Staubli VAL3: Shell.dtx

bool b1 = true
bool b2 = true
bool bExit
bool bInit
bool bListRefresh = true
bool bPause
bool bRobAtStP
bool bUserRefresh = true
dio distart = {link=usrIn0}
dio distop = {link=usrIn1}
dio ditab = {link=BasicIO-1\%I1}
dio dixi = {link=BasicIO-1\%I0}
dio dochui = {link=BasicIO-1\%Q0}
dio doxi = {link=BasicIO-1\%Q1}
frame f1 = {x=118.3, y=-256.27, z=-98.22, rx=-0.18, ry=0.05, rz=179.93, fatherId=world[0]}
frame fFrmTemp = {x=480, y=75, z=-95.95, rx=5, ry=0, rz=-93, fatherId=world[0]}
frame frmaster = {x=480, y=75, z=-95.95, rx=5, rz=-93, fatherId=world[0]}
jointRx jXieLiao = {j1=-98.995401, j2=73.939591, j3=22.369301, j4=-0.0214, j5=83.505129, j6=-98.792613}
jointRx jbegin = {j1=-36.809158, j2=6.473103, j3=115.475326, j4=0.67904, j5=57.498227, j6=-129.910351}
jointRx jchack = {j1=-93.592762, j2=7.01746, j3=116.913403, j4=-0.052986, j5=55.884155, j6=86.700695}
jointRx jend = {j1=-46.642796, j2=10.279087, j3=109.084102, j4=6.799386, j5=57.689141, j6=-43.494821}
jointRx jready = {j1=-93.60071, j2=14.149819, j3=120.13944, j4=-0.061569, j5=45.526614, j6=86.705521}
jointRx jstart = {j1=-93.593066, j2=7.017202, j3=116.913452, j4=-0.053086, j5=55.884413, j6=86.699801}
mdesc m1
mdesc mSuDu[3]
  [0] = {leave=0.5, reach=0.5}
  [1] = {accel=25, vel=50, decel=25, leave=0.5, reach=0.5}
  [2] = {leave=0.5, reach=0.5}
num n0 = 1
num n1 = 2
num n2
num nBeltLifeTime = 1000
num nPY
num nPYB
num nPYC
num nPYtest
num nPage
num nSelected
num nSize = 314
num nc
num ndemo = 314
num ni
pointRx p1 = {x=0.29, y=-0.21, z=62.49, rx=-180, rz=179.71, fatherId=f1[0]}
pointRx p2 = {x=0.29, y=-0.21, z=-0.5, rx=-180, rz=179.71, fatherId=f1[0]}
pointRx p3 = {x=-135.757719, y=-14.921956, z=109.991113, rx=0.040194, ry=-179.896326, rz=-0.477597, fatherId=f1[0]}
pointRx p4 = {x=-342.629435, y=-93.502982, z=80.205763, rx=0.07546, ry=-170.514293, rz=20.52476, fatherId=f1[0]}
pointRx p5 = {x=-343.525561, y=-394.240354, z=80.654544, rx=173.283811, ry=-0.218212, rz=-67.079827, fatherId=f1[0]}
pointRx pTemp = {x=-72.136382, y=-5.208147, z=99.387825, rx=179.99914, ry=-2.97245, rz=-27.003129, shoulder=lefty, elbow=epositive, wrist=wpositive, fatherId=fFrmTemp[0]}
pointRx pXieLiao[2]
  [0] = {x=530.900904, y=-168.692362, z=119.392812, rx=179.999348, ry=-0.000559, rz=86.125781, fatherId=f1[0]}
  [1] = {x=530.900895, y=-168.692364, z=88.853022, rx=179.999359, ry=-0.000487, rz=86.125781, fatherId=f1[0]}
pointRx pdemo[900]
  [0] = {x=-72.139316, y=-5.205403, z=114.395923, rx=-179.99945, ry=-2.972824, rz=-27.002856, shoulder=lefty, elbow=epositive, wrist=wpositive, fatherId=frmaster[0]}
  [1] = {x=-72.141191, y=-5.207684, z=109.390059, rx=179.999959, ry=-2.973162, rz=-27.002729, shoulder=lefty, elbow=epositive, wrist=wpositive, fatherId=frmaster[0]}
  [2] = {x=-72.136382, y=-5.208147, z=99.387825, rx=179.99914, ry=-2.97245, rz=-27.003129, shoulder=lefty, elbow=epositive, wrist=wpositive, fatherId=frmaster[0]}
  [3] = {x=-68.975889, y=-15.06218, z=100.784201, rx=179.999892, ry=-4.176426, rz=-34.805987, shoulder=lefty, elbow=epositive, wrist=wpositive, fatherId=frmaster[0]}
  [4] = {x=-62.859726, y=-25.676052, z=102.773744, rx=179.999165, ry=-6.140672, rz=-43.339442, shoulder=lefty, elbow=epositive, wrist=wpositive, fatherId=frmaster[0]}
  [5] = {x=-58.874108, y=-29.961824, z=104.027701, rx=179.999797, ry=-7.513724, rz=-46.917099, shoulder=lefty, elbow=epositive, wrist=wpositive, fatherId=frmaster[0]}
  [6] = {x=-54.218, y=-33.710091, z=105.454934, rx=179.999588, ry=-9.225876, rz=-50.125341, shoulder=lefty, elbow=epositive, wrist=wpositive, fatherId=frmaster[0]}
  [7] = {x=-48.8955, y=-37.045292, z=106.967933, rx=179.999506, ry=-11.262628, rz=-53.058248, shoulder=lefty, elbow=epositive, wrist=wpositive, fatherId=frmaster[0]}
  [8] = {x=-42.768943, y=-40.048852, z=108.527677, rx=179.999261, ry=-13.708147, rz=-55.767693, shoulder=lefty, elbow=epositive, wrist=wpositive, fatherId=frmaster[0]}
  [9] = {x=-35.863349, y=-42.736386, z=110.015011, rx=179.999729, ry=-16.552892, rz=-58.259195, shoulder=lefty, elbow=epositive, wrist=wpositive, fatherId=frmaster[0]}
  [10] = {x=-32.052155, y=-43.961424, z=110.710133, rx=-179.999047, ry=-18.162895, rz=-59.423084, shoulder=lefty, elbow=epositive, wrist=wpositive, fatherId=frmaster[0]}
  [11] = {x=-27.998338, y=-45.113393, z=111.337723, rx=179.999655, ry=-19.903876, rz=-60.529866, shoulder=lefty, elbow=epositive, wrist=wpositive, fatherId=frmaster[0]}
  [12] = {x=-23.770579, y=-46.150343, z=111.884468, rx=179.999725, ry=-21.757032, rz=-61.544546, shoulder=lefty, elbow=epositive, wrist=wpositive, fatherId=frmaster[0]}
  [13] = {x=-19.355958, y=-47.062466, z=112.34637, rx=179.999568, ry=-23.731431, rz=-62.455355, shoulder=lefty, elbow=epositive, wrist=wpositive, fatherId=frmaster[0]}
  [14] = {x=-14.798675, y=-47.863527, z=112.678078, rx=179.999356, ry=-25.809627, rz=-63.271003, shoulder=lefty, elbow=epositive, wrist=wpositive, fatherId=frmaster[0]}
  [15] = {x=-10.132044, y=-48.569614, z=112.872483, rx=179.999563, ry=-27.969963, rz=-64.002263, shoulder=lefty, elbow=epositive, wrist=wpositive, fatherId=frmaster[0]}
  [16] = {x=-5.340054, y=-49.191372, z=112.899752, rx=179.999359, ry=-30.221279, rz=-64.662655, shoulder=lefty, elbow=epositive, wrist=wpositive, fatherId=frmaster[0]}
  [17] = {x=-0.497659, y=-49.744484, z=112.745007, rx=179.997593, ry=-32.530564, rz=-65.260267, shoulder=lefty, elbow=epositive, wrist=wpositive, fatherId=frmaster[0]}
  [18] = {x=4.355318, y=-50.231725, z=112.407987, rx=179.998323, ry=-34.873687, rz=-65.799828, shoulder=lefty, elbow=epositive, wrist=wpositive, fatherId=frmaster[0]}
  [19] = {x=9.191912, y=-50.662039, z=111.876558, rx=179.999421, ry=-37.237015, rz=-66.289828, shoulder=lefty, elbow=epositive, wrist=wpositive, fatherId=frmaster[0]}
  [20] = {x=14.065883, y=-51.011691, z=111.155805, rx=179.998913, ry=-39.669144, rz=-66.696703, shoulder=lefty, elbow=epositive, wrist=wpositive, fatherId=frmaster[0]}
  [21] = {x=18.80483, y=-51.332378, z=110.24932, rx=179.997399, ry=-42.066597, rz=-67.075927, shoulder=lefty, elbow=epositive, wrist=wpositive, fatherId=frmaster[0]}
  [22] = {x=23.272914, y=-51.627115, z=109.187587, rx=179.998413, ry=-44.352778, rz=-67.433341, shoulder=lefty, elbow=epositive, wrist=wpositive, fatherId=frmaster[0]}
  [23] = {x=27.490839, y=-51.903449, z=107.99836, rx=179.9978, ry=-46.542828, rz=-67.774892, shoulder=lefty, elbow=epositive, wrist=wpositive, fatherId=frmaster[0]}
  [24] = {x=31.656111, y=-52.09758, z=106.686347, rx=179.997482, ry=-48.76331, rz=-68.024803, shoulder=lefty, elbow=epositive, wrist=wpositive, fatherId=frmaster[0]}
  [25] = {x=35.832908, y=-52.268838, z=105.191277, rx=179.998026, ry=-51.03047, rz=-68.257472, shoulder=lefty, elbow=epositive, wrist=wpositive, fatherId=frmaster[0]}
  [26] = {x=40.028913, y=-52.432584, z=103.494456, rx=179.99633, ry=-53.350485, rz=-68.477247, shoulder=lefty, elbow=epositive, wrist=wpositive, fatherId=frmaster[0]}
  [27] = {x=44.046496, y=-52.586328, z=101.6722, rx=179.996899, ry=-55.612206, rz=-68.689407, shoulder=lefty, elbow=epositive, wrist=wpositive, fatherId=frmaster[0]}
  [28] = {x=47.812574, y=-52.649532, z=99.828642, rx=179.995594, ry=-57.811363, rz=-68.802993, shoulder=lefty, elbow=epositive, wrist=wpositive, fatherId=frmaster[0]}
  [29] = {x=51.331952, y=-52.69796, z=97.929572, rx=179.997025, ry=-59.911141, rz=-68.903832, shoulder=lefty, elbow=epositive, wrist=wpositive, fatherId=frmaster[0]}
  [30] = {x=55.491329, y=-52.735941, z=95.502133, rx=179.997027, ry=-62.4448, rz=-68.990371, shoulder=lefty, elbow=epositive, wrist=wpositive, fatherId=frmaster[0]}
  [31] = {x=57.921659, y=-52.752353, z=93.971659, rx=179.995202, ry=-63.949927, rz=-69.033741, shoulder=lefty, elbow=epositive, wrist=wpositive, fatherId=frmaster[0]}
  [32] = {x=60.537153, y=-52.77071, z=92.230547, rx=179.995383, ry=-65.598259, rz=-69.077786, shoulder=lefty, elbow=epositive, wrist=wpositive, fatherId=frmaster[0]}
  [33] = {x=56.995232, y=-51.826133, z=95.154639, rx=179.99741, ry=-63.625523, rz=-67.991265, shoulder=lefty, elbow=epositive, wrist=wpositive, fatherId=frmaster[0]}
  [34] = {x=53.839502, y=-50.855589, z=97.641731, rx=179.998709, ry=-61.953126, rz=-66.894176, shoulder=lefty, elbow=epositive, wrist=wpositive, fatherId=frmaster[0]}
  [35] = {x=51.097923, y=-49.850634, z=99.754671, rx=179.995572, ry=-60.579202, rz=-65.784532, shoulder=lefty, elbow=epositive, wrist=wpositive, fatherId=frmaster[0]}
  [36] = {x=48.698616, y=-48.800611, z=101.606549, rx=179.998668, ry=-59.430163, rz=-64.64955, shoulder=lefty, elbow=epositive, wrist=wpositive, fatherId=frmaster[0]}
  [37] = {x=44.979407, y=-46.331543, z=104.677115, rx=179.996454, ry=-57.904138, rz=-62.075166, shoulder=lefty, elbow=epositive, wrist=wpositive, fatherId=frmaster[0]}
  [38] = {x=41.185661, y=-43.702, z=107.55876, rx=179.997987, ry=-56.386554, rz=-59.438386, shoulder=lefty, elbow=epositive, wrist=wpositive, fatherId=frmaster[0]}
  [39] = {x=38.104587, y=-40.71475, z=110.038066, rx=179.99707, ry=-55.338217, rz=-56.569911, shoulder=lefty, elbow=epositive, wrist=wpositive, fatherId=frmaster[0]}
  [40] = {x=35.18463, y=-37.4952, z=112.304852, rx=179.997372, ry=-54.390812, rz=-53.584816, shoulder=lefty, elbow=epositive, wrist=wpositive, fatherId=frmaster[0]}
  [41] = {x=32.57611, y=-34.062936, z=114.327999, rx=179.997864, ry=-53.602083, rz=-50.509719, shoulder=lefty, elbow=epositive, wrist=wpositive, fatherId=frmaster[0]}
  [42] = {x=30.347907, y=-30.459195, z=116.077336, rx=179.996571, ry=-52.98833, rz=-47.372839, shoulder=lefty, elbow=epositive, wrist=wpositive, fatherId=frmaster[0]}
  [43] = {x=27.630594, y=-26.739916, z=117.787752, rx=179.997373, ry=-52.090979, rz=-44.216779, shoulder=lefty, elbow=epositive, wrist=wpositive, fatherId=frmaster[0]}
  [44] = {x=25.387415, y=-22.814503, z=119.214392, rx=179.997777, ry=-51.397674, rz=-40.964839, shoulder=lefty, elbow=epositive, wrist=wpositive, fatherId=frmaster[0]}
  [45] = {x=21.907259, y=-18.829629, z=120.677376, rx=179.997241, ry=-50.051737, rz=-37.723844, shoulder=lefty, elbow=epositive, wrist=wpositive, fatherId=frmaster[0]}
  [46] = {x=18.976892, y=-14.698385, z=121.811971, rx=179.997739, ry=-48.928716, rz=-34.417507, shoulder=lefty, elbow=epositive, wrist=wpositive, fatherId=frmaster[0]}
  [47] = {x=15.189076, y=-10.641411, z=122.819382, rx=179.998604, ry=-47.333182, rz=-31.199476, shoulder=lefty, elbow=epositive, wrist=wpositive, fatherId=frmaster[0]}
  [48] = {x=12.160817, y=-6.550912, z=123.480224, rx=179.998107, ry=-46.04514, rz=-27.978628, shoulder=lefty, elbow=epositive, wrist=wpositive, fatherId=frmaster[0]}
  [49] = {x=9.062094, y=-2.446034, z=123.915808, rx=179.998654, ry=-44.656407, rz=-24.757058, shoulder=lefty, elbow=epositive, wrist=wpositive, fatherId=frmaster[0]}
  [50] = {x=6.937856, y=1.678803, z=124.07243, rx=179.998216, ry=-43.654199, rz=-21.525314, shoulder=lefty, elbow=epositive, wrist=wpositive, fatherId=frmaster[0]}
  [51] = {x=5.582997, y=5.684193, z=124.012721, rx=179.998101, ry=-42.934062, rz=-18.365961, shoulder=lefty, elbow=epositive, wrist=wpositive, fatherId=frmaster[0]}
  [52] = {x=5.181143, y=9.295156, z=123.790887, rx=179.998253, ry=-42.608226, rz=-15.478968, shoulder=lefty, elbow=epositive, wrist=wpositive, fatherId=frmaster[0]}
  [53] = {x=6.162431, y=12.507722, z=123.420614, rx=179.998637, ry=-42.889469, rz=-12.857822, shoulder=lefty, elbow=epositive, wrist=wpositive, fatherId=frmaster[0]}
  [54] = {x=7.857103, y=15.304792, z=122.959895, rx=179.999415, ry=-43.485371, rz=-10.519163, shoulder=lefty, elbow=epositive, wrist=wpositive, fatherId=frmaster[0]}
  [55] = {x=3.99638, y=15.043622, z=123.176677, rx=179.997318, ry=-41.674084, rz=-10.720178, shoulder=lefty, elbow=epositive, wrist=wpositive, fatherId=frmaster[0]}
  [56] = {x=0.076533, y=14.77642, z=123.28561, rx=179.999597, ry=-39.835796, rz=-10.928558, shoulder=lefty, elbow=epositive, wrist=wpositive, fatherId=frmaster[0]}
  [57] = {x=-3.902392, y=14.490264, z=123.256768, rx=179.998802, ry=-37.973068, rz=-11.148301, shoulder=lefty, elbow=epositive, wrist=wpositive, fatherId=frmaster[0]}
  [58] = {x=-7.919724, y=14.195071, z=123.100201, rx=-179.999948, ry=-36.090049, rz=-11.376972, shoulder=lefty, elbow=epositive, wrist=wpositive, fatherId=frmaster[0]}
  [59] = {x=-11.781305, y=13.882374, z=122.822648, rx=179.999835, ry=-34.281196, rz=-11.618916, shoulder=lefty, elbow=epositive, wrist=wpositive, fatherId=frmaster[0]}
  [60] = {x=-15.483544, y=13.561811, z=122.438491, rx=179.998456, ry=-32.542349, rz=-11.865332, shoulder=lefty, elbow=epositive, wrist=wpositive, fatherId=frmaster[0]}
  [61] = {x=-19.01741, y=13.241039, z=121.965321, rx=179.998614, ry=-30.873858, rz=-12.11299, shoulder=lefty, elbow=epositive, wrist=wpositive, fatherId=frmaster[0]}
  [62] = {x=-22.396274, y=12.91462, z=121.416049, rx=179.999262, ry=-29.273631, rz=-12.364904, shoulder=lefty, elbow=epositive, wrist=wpositive, fatherId=frmaster[0]}
  [63] = {x=-25.613574, y=12.577452, z=120.800174, rx=179.999931, ry=-27.738912, rz=-12.627295, shoulder=lefty, elbow=epositive, wrist=wpositive, fatherId=frmaster[0]}
  [64] = {x=-28.708425, y=12.226522, z=120.125533, rx=179.998558, ry=-26.259538, rz=-12.895843, shoulder=lefty, elbow=epositive, wrist=wpositive, fatherId=frmaster[0]}
  [65] = {x=-34.488439, y=11.514031, z=118.631959, rx=179.999255, ry=-23.46879, rz=-13.449377, shoulder=lefty, elbow=epositive, wrist=wpositive, fatherId=frmaster[0]}
  [66] = {x=-39.717604, y=10.760933, z=117.019852, rx=179.999112, ry=-20.908672, rz=-14.032246, shoulder=lefty, elbow=epositive, wrist=wpositive, fatherId=frmaster[0]}
  [67] = {x=-44.357262, y=10.000083, z=115.366462, rx=-179.999814, ry=-18.600675, rz=-14.622901, shoulder=lefty, elbow=epositive, wrist=wpositive, fatherId=frmaster[0]}
  [68] = {x=-48.465875, y=9.222145, z=113.704261, rx=179.999952, ry=-16.51928, rz=-15.22769, shoulder=lefty, elbow=epositive, wrist=wpositive, fatherId=frmaster[0]}
  [69] = {x=-52.032354, y=8.458188, z=112.118175, rx=179.998905, ry=-14.683899, rz=-15.823133, shoulder=lefty, elbow=epositive, wrist=wpositive, fatherId=frmaster[0]}
  [70] = {x=-55.116158, y=7.71911, z=110.629883, rx=-179.999954, ry=-13.066095, rz=-16.404411, shoulder=lefty, elbow=epositive, wrist=wpositive, fatherId=frmaster[0]}
  [71] = {x=-57.708156, y=7.045592, z=109.275583, rx=179.999755, ry=-11.675002, rz=-16.940666, shoulder=lefty, elbow=epositive, wrist=wpositive, fatherId=frmaster[0]}
  [72] = {x=-62.051935, y=5.747157, z=106.795298, rx=-179.999723, ry=-9.281904, rz=-17.979557, shoulder=lefty, elbow=epositive, wrist=wpositive, fatherId=frmaster[0]}
  [73] = {x=-65.470295, y=4.550856, z=104.61812, rx=179.999718, ry=-7.320707, rz=-18.952356, shoulder=lefty, elbow=epositive, wrist=wpositive, fatherId=frmaster[0]}
  [74] = {x=-69.996671, y=2.629302, z=101.343766, rx=-179.999852, ry=-4.53887, rz=-20.57499, shoulder=lefty, elbow=epositive, wrist=wpositive, fatherId=frmaster[0]}
  [75] = {x=-70.001872, y=2.626567, z=111.346309, rx=179.999708, ry=-4.53945, rz=-20.575404, shoulder=lefty, elbow=epositive, wrist=wpositive, fatherId=frmaster[0]}
  [76] = {x=-69.994182, y=2.628439, z=116.339052, rx=179.999809, ry=-4.538758, rz=-20.574443, shoulder=lefty, elbow=epositive, wrist=wpositive, fatherId=frmaster[0]}
  [77] = {x=-69.238992, y=2.628498, z=125.877606, rx=-179.999522, ry=-4.539031, rz=-20.574278, shoulder=lefty, elbow=epositive, wrist=wpositive, fatherId=frmaster[0]}
  [78] = {x=-71.822664, y=-5.297555, z=123.895608, rx=0.000097, ry=-177.027023, rz=-27.002375, shoulder=lefty, elbow=epositive, wrist=wpositive, fatherId=frmaster[0]}
  [79] = {x=-72.317273, y=-5.29621, z=114.405164, rx=0.00055, ry=-177.027176, rz=-27.002856, shoulder=lefty, elbow=epositive, wrist=wpositive, fatherId=frmaster[0]}
  [80] = {x=-72.319148, y=-5.298491, z=109.399302, rx=-0.000041, ry=-177.026838, rz=-27.002729, shoulder=lefty, elbow=epositive, wrist=wpositive, fatherId=frmaster[0]}
  [81] = {x=-72.314338, y=-5.298955, z=99.397067, rx=-0.00086, ry=-177.02755, rz=-27.003129, shoulder=lefty, elbow=epositive, wrist=wpositive, fatherId=frmaster[0]}
  [82] = {x=-69.13967, y=-15.17634, z=100.796161, rx=-0.000108, ry=-175.823574, rz=-34.805987, shoulder=lefty, elbow=epositive, wrist=wpositive, fatherId=frmaster[0]}
  [83] = {x=-63.004351, y=-25.813316, z=102.789306, rx=-0.000835, ry=-173.859328, rz=-43.339442, shoulder=lefty, elbow=epositive, wrist=wpositive, fatherId=frmaster[0]}
  [84] = {x=-59.009546, y=-30.107897, z=104.045565, rx=-0.000203, ry=-172.486276, rz=-46.917099, shoulder=lefty, elbow=epositive, wrist=wpositive, fatherId=frmaster[0]}
  [85] = {x=-54.344563, y=-33.86358, z=105.475492, rx=-0.000412, ry=-170.774124, rz=-50.125341, shoulder=lefty, elbow=epositive, wrist=wpositive, fatherId=frmaster[0]}
  [86] = {x=-49.013385, y=-37.205141, z=106.99141, rx=-0.000494, ry=-168.737372, rz=-53.058248, shoulder=lefty, elbow=epositive, wrist=wpositive, fatherId=frmaster[0]}
  [87] = {x=-42.878248, y=-40.214205, z=108.554341, rx=-0.000739, ry=-166.291853, rz=-55.767693, shoulder=lefty, elbow=epositive, wrist=wpositive, fatherId=frmaster[0]}
  [88] = {x=-35.964204, y=-42.906473, z=110.044988, rx=-0.000271, ry=-163.447108, rz=-58.259195, shoulder=lefty, elbow=epositive, wrist=wpositive, fatherId=frmaster[0]}
  [89] = {x=-32.148825, y=-44.133614, z=110.741844, rx=0.000953, ry=-161.837105, rz=-59.423084, shoulder=lefty, elbow=epositive, wrist=wpositive, fatherId=frmaster[0]}
  [90] = {x=-28.090855, y=-45.287515, z=111.371222, rx=-0.000345, ry=-160.096124, rz=-60.529866, shoulder=lefty, elbow=epositive, wrist=wpositive, fatherId=frmaster[0]}
  [91] = {x=-23.859086, y=-46.326181, z=111.919792, rx=-0.000275, ry=-158.242968, rz=-61.544546, shoulder=lefty, elbow=epositive, wrist=wpositive, fatherId=frmaster[0]}
  [92] = {x=-19.440625, y=-47.239796, z=112.383594, rx=-0.000432, ry=-156.268569, rz=-62.455355, shoulder=lefty, elbow=epositive, wrist=wpositive, fatherId=frmaster[0]}
  [93] = {x=-14.879656, y=-48.042155, z=112.717245, rx=-0.000644, ry=-154.190373, rz=-63.271003, shoulder=lefty, elbow=epositive, wrist=wpositive, fatherId=frmaster[0]}
  [94] = {x=-10.209471, y=-48.749376, z=112.913601, rx=-0.000437, ry=-152.030037, rz=-64.002263, shoulder=lefty, elbow=epositive, wrist=wpositive, fatherId=frmaster[0]}
  [95] = {x=-5.414011, y=-49.372132, z=112.942835, rx=-0.000641, ry=-149.778721, rz=-64.662655, shoulder=lefty, elbow=epositive, wrist=wpositive, fatherId=frmaster[0]}
  [96] = {x=-0.568227, y=-49.926126, z=112.790024, rx=-0.002407, ry=-147.469436, rz=-65.260267, shoulder=lefty, elbow=epositive, wrist=wpositive, fatherId=frmaster[0]}
  [97] = {x=4.288056, y=-50.414147, z=112.454869, rx=-0.001677, ry=-145.126313, rz=-65.799828, shoulder=lefty, elbow=epositive, wrist=wpositive, fatherId=frmaster[0]}
  [98] = {x=9.127885, y=-50.845157, z=111.925225, rx=-0.000579, ry=-142.762985, rz=-66.289828, shoulder=lefty, elbow=epositive, wrist=wpositive, fatherId=frmaster[0]}
  [99] = {x=14.004981, y=-51.195375, z=111.206315, rx=-0.001087, ry=-140.330856, rz=-66.696703, shoulder=lefty, elbow=epositive, wrist=wpositive, fatherId=frmaster[0]}
  [100] = {x=18.746998, y=-51.51658, z=110.301523, rx=-0.002601, ry=-137.933403, rz=-67.075927, shoulder=lefty, elbow=epositive, wrist=wpositive, fatherId=frmaster[0]}
  [101] = {x=23.218033, y=-51.811801, z=109.241247, rx=-0.001587, ry=-135.647222, rz=-67.433341, shoulder=lefty, elbow=epositive, wrist=wpositive, fatherId=frmaster[0]}
  [102] = {x=27.438806, y=-52.088588, z=108.05328, rx=-0.0022, ry=-133.457172, rz=-67.774892, shoulder=lefty, elbow=epositive, wrist=wpositive, fatherId=frmaster[0]}
  [103] = {x=31.606778, y=-52.283047, z=106.742635, rx=-0.002518, ry=-131.23669, rz=-68.024803, shoulder=lefty, elbow=epositive, wrist=wpositive, fatherId=frmaster[0]}
  [104] = {x=35.786314, y=-52.454607, z=105.248884, rx=-0.001974, ry=-128.96953, rz=-68.257472, shoulder=lefty, elbow=epositive, wrist=wpositive, fatherId=frmaster[0]}
  [105] = {x=39.985115, y=-52.618635, z=103.553336, rx=-0.00367, ry=-126.649515, rz=-68.477247, shoulder=lefty, elbow=epositive, wrist=wpositive, fatherId=frmaster[0]}
  [106] = {x=44.005444, y=-52.77265, z=101.732192, rx=-0.003101, ry=-124.387794, rz=-68.689407, shoulder=lefty, elbow=epositive, wrist=wpositive, fatherId=frmaster[0]}
  [107] = {x=47.774051, y=-52.835995, z=99.889857, rx=-0.004406, ry=-122.188637, rz=-68.802993, shoulder=lefty, elbow=epositive, wrist=wpositive, fatherId=frmaster[0]}
  [108] = {x=51.295861, y=-52.884553, z=97.991868, rx=-0.002975, ry=-120.088859, rz=-68.903832, shoulder=lefty, elbow=epositive, wrist=wpositive, fatherId=frmaster[0]}
  [109] = {x=55.458158, y=-52.922641, z=95.565714, rx=-0.002973, ry=-117.5552, rz=-68.990371, shoulder=lefty, elbow=epositive, wrist=wpositive, fatherId=frmaster[0]}
  [110] = {x=57.890231, y=-52.939106, z=94.035968, rx=-0.004798, ry=-116.050073, rz=-69.033741, shoulder=lefty, elbow=epositive, wrist=wpositive, fatherId=frmaster[0]}
  [111] = {x=60.507647, y=-52.957518, z=92.295603, rx=-0.004617, ry=-114.401741, rz=-69.077786, shoulder=lefty, elbow=epositive, wrist=wpositive, fatherId=frmaster[0]}
  [112] = {x=56.961937, y=-52.011555, z=95.221795, rx=-0.00259, ry=-116.374477, rz=-67.991265, shoulder=lefty, elbow=epositive, wrist=wpositive, fatherId=frmaster[0]}
  [113] = {x=53.802599, y=-51.039544, z=97.711004, rx=-0.001291, ry=-118.046874, rz=-66.894176, shoulder=lefty, elbow=epositive, wrist=wpositive, fatherId=frmaster[0]}
  [114] = {x=51.057627, y=-50.03303, z=99.82614, rx=-0.004428, ry=-119.420798, rz=-65.784532, shoulder=lefty, elbow=epositive, wrist=wpositive, fatherId=frmaster[0]}
  [115] = {x=48.655065, y=-48.981351, z=101.680283, rx=-0.001332, ry=-120.569837, rz=-64.64955, shoulder=lefty, elbow=epositive, wrist=wpositive, fatherId=frmaster[0]}
  [116] = {x=44.929641, y=-46.50825, z=104.756473, rx=-0.003546, ry=-122.095862, rz=-62.075166, shoulder=lefty, elbow=epositive, wrist=wpositive, fatherId=frmaster[0]}
  [117] = {x=41.129365, y=-43.874214, z=107.643455, rx=-0.002013, ry=-123.613446, rz=-59.438386, shoulder=lefty, elbow=epositive, wrist=wpositive, fatherId=frmaster[0]}
  [118] = {x=38.041922, y=-40.881657, z=110.128703, rx=-0.00293, ry=-124.661783, rz=-56.569911, shoulder=lefty, elbow=epositive, wrist=wpositive, fatherId=frmaster[0]}
  [119] = {x=35.115501, y=-37.656143, z=112.401385, rx=-0.002628, ry=-125.609188, rz=-53.584816, shoulder=lefty, elbow=epositive, wrist=wpositive, fatherId=frmaster[0]}
  [120] = {x=32.500637, y=-34.217279, z=114.430381, rx=-0.002136, ry=-126.397917, rz=-50.509719, shoulder=lefty, elbow=epositive, wrist=wpositive, fatherId=frmaster[0]}
  [121] = {x=30.266372, y=-30.606344, z=116.1855, rx=-0.003429, ry=-127.01167, rz=-47.372839, shoulder=lefty, elbow=epositive, wrist=wpositive, fatherId=frmaster[0]}
  [122] = {x=27.542523, y=-26.879386, z=117.900853, rx=-0.002627, ry=-127.909021, rz=-44.216779, shoulder=lefty, elbow=epositive, wrist=wpositive, fatherId=frmaster[0]}
  [123] = {x=25.29319, y=-22.945618, z=119.332421, rx=-0.002223, ry=-128.602326, rz=-40.964839, shoulder=lefty, elbow=epositive, wrist=wpositive, fatherId=frmaster[0]}
  [124] = {x=21.805684, y=-18.951994, z=120.798657, rx=-0.002759, ry=-129.948263, rz=-37.723844, shoulder=lefty, elbow=epositive, wrist=wpositive, fatherId=frmaster[0]}
  [125] = {x=18.868495, y=-14.811424, z=121.936359, rx=-0.002261, ry=-131.071284, rz=-34.417507, shoulder=lefty, elbow=epositive, wrist=wpositive, fatherId=frmaster[0]}
  [126] = {x=15.073134, y=-10.745011, z=122.945176, rx=-0.001396, ry=-132.666818, rz=-31.199476, shoulder=lefty, elbow=epositive, wrist=wpositive, fatherId=frmaster[0]}
  [127] = {x=12.038223, y=-6.644737, z=123.607377, rx=-0.001893, ry=-133.95486, rz=-27.978628, shoulder=lefty, elbow=epositive, wrist=wpositive, fatherId=frmaster[0]}
  [128] = {x=8.932903, y=-2.529785, z=124.043461, rx=-0.001346, ry=-135.343593, rz=-24.757058, shoulder=lefty, elbow=epositive, wrist=wpositive, fatherId=frmaster[0]}
  [129] = {x=6.803245, y=1.605425, z=124.200864, rx=-0.001784, ry=-136.345801, rz=-21.525314, shoulder=lefty, elbow=epositive, wrist=wpositive, fatherId=frmaster[0]}
  [130] = {x=5.444027, y=5.62118, z=124.142015, rx=-0.001899, ry=-137.065938, rz=-18.365961, shoulder=lefty, elbow=epositive, wrist=wpositive, fatherId=frmaster[0]}
  [131] = {x=5.039282, y=9.241783, z=123.921374, rx=-0.001747, ry=-137.391774, rz=-15.478968, shoulder=lefty, elbow=epositive, wrist=wpositive, fatherId=frmaster[0]}
  [132] = {x=6.019572, y=12.463219, z=123.553319, rx=-0.001363, ry=-137.110531, rz=-12.857822, shoulder=lefty, elbow=epositive, wrist=wpositive, fatherId=frmaster[0]}
  [133] = {x=7.714432, y=15.26828, z=123.095216, rx=-0.000585, ry=-136.514629, rz=-10.519163, shoulder=lefty, elbow=epositive, wrist=wpositive, fatherId=frmaster[0]}
  [134] = {x=3.849599, y=15.006425, z=123.307336, rx=-0.002682, ry=-138.325916, rz=-10.720178, shoulder=lefty, elbow=epositive, wrist=wpositive, fatherId=frmaster[0]}
  [135] = {x=-0.074258, y=14.738504, z=123.411405, rx=-0.000403, ry=-140.164204, rz=-10.928558, shoulder=lefty, elbow=epositive, wrist=wpositive, fatherId=frmaster[0]}
  [136] = {x=-4.057077, y=14.451596, z=123.377505, rx=-0.001198, ry=-142.026932, rz=-11.148301, shoulder=lefty, elbow=epositive, wrist=wpositive, fatherId=frmaster[0]}
  [137] = {x=-8.078166, y=14.155618, z=123.215697, rx=0.000052, ry=-143.909951, rz=-11.376972, shoulder=lefty, elbow=epositive, wrist=wpositive, fatherId=frmaster[0]}
  [138] = {x=-11.943175, y=13.842094, z=122.932991, rx=-0.000165, ry=-145.718804, rz=-11.618916, shoulder=lefty, elbow=epositive, wrist=wpositive, fatherId=frmaster[0]}
  [139] = {x=-15.64854, y=13.520691, z=122.543778, rx=-0.001544, ry=-147.457651, rz=-11.865332, shoulder=lefty, elbow=epositive, wrist=wpositive, fatherId=frmaster[0]}
  [140] = {x=-19.185248, y=13.199074, z=122.065667, rx=-0.001386, ry=-149.126142, rz=-12.11299, shoulder=lefty, elbow=epositive, wrist=wpositive, fatherId=frmaster[0]}
  [141] = {x=-22.566686, y=12.871794, z=121.511578, rx=-0.000738, ry=-150.726369, rz=-12.364904, shoulder=lefty, elbow=epositive, wrist=wpositive, fatherId=frmaster[0]}
  [142] = {x=-25.786308, y=12.53373, z=120.891011, rx=-0.000069, ry=-152.261088, rz=-12.627295, shoulder=lefty, elbow=epositive, wrist=wpositive, fatherId=frmaster[0]}
  [143] = {x=-28.883261, y=12.181888, z=120.21179, rx=-0.001442, ry=-153.740462, rz=-12.895843, shoulder=lefty, elbow=epositive, wrist=wpositive, fatherId=frmaster[0]}
  [144] = {x=-34.666863, y=11.467515, z=118.709425, rx=-0.000745, ry=-156.53121, rz=-13.449377, shoulder=lefty, elbow=epositive, wrist=wpositive, fatherId=frmaster[0]}
  [145] = {x=-39.898859, y=10.71244, z=117.089099, rx=-0.000888, ry=-159.091328, rz=-14.032246, shoulder=lefty, elbow=epositive, wrist=wpositive, fatherId=frmaster[0]}
  [146] = {x=-44.540675, y=9.949592, z=115.42819, rx=0.000186, ry=-161.399325, rz=-14.622901, shoulder=lefty, elbow=epositive, wrist=wpositive, fatherId=frmaster[0]}
  [147] = {x=-48.650887, y=9.169614, z=113.759132, rx=-0.000048, ry=-163.48072, rz=-15.22769, shoulder=lefty, elbow=epositive, wrist=wpositive, fatherId=frmaster[0]}
  [148] = {x=-52.218491, y=8.403656, z=112.166953, rx=-0.001095, ry=-165.316101, rz=-15.823133, shoulder=lefty, elbow=epositive, wrist=wpositive, fatherId=frmaster[0]}
  [149] = {x=-55.303049, y=7.662627, z=110.673258, rx=0.000046, ry=-166.933905, rz=-16.404411, shoulder=lefty, elbow=epositive, wrist=wpositive, fatherId=frmaster[0]}
  [150] = {x=-57.895519, y=6.987316, z=109.314299, rx=-0.000245, ry=-168.324998, rz=-16.940666, shoulder=lefty, elbow=epositive, wrist=wpositive, fatherId=frmaster[0]}
  [151] = {x=-62.239678, y=5.685421, z=106.825981, rx=0.000277, ry=-170.718096, rz=-17.979557, shoulder=lefty, elbow=epositive, wrist=wpositive, fatherId=frmaster[0]}
  [152] = {x=-65.65791, y=4.485899, z=104.642223, rx=-0.000282, ry=-172.679293, rz=-18.952356, shoulder=lefty, elbow=epositive, wrist=wpositive, fatherId=frmaster[0]}
  [153] = {x=-70.183327, y=2.559015, z=101.358584, rx=0.000148, ry=-175.46113, rz=-20.57499, shoulder=lefty, elbow=epositive, wrist=wpositive, fatherId=frmaster[0]}
  [154] = {x=-70.188527, y=2.556279, z=111.361129, rx=-0.000292, ry=-175.46055, rz=-20.575404, shoulder=lefty, elbow=epositive, wrist=wpositive, fatherId=frmaster[0]}
  [155] = {x=-70.180838, y=2.558154, z=116.353869, rx=-0.000191, ry=-175.461242, rz=-20.574443, shoulder=lefty, elbow=epositive, wrist=wpositive, fatherId=frmaster[0]}
  [156] = {x=-69.425648, y=2.558214, z=125.892424, rx=0.000478, ry=-175.460969, rz=-20.574278, shoulder=lefty, elbow=epositive, wrist=wpositive, fatherId=frmaster[0]}
  [157] = {x=-69.427023, y=-2.562467, z=125.884136, rx=-0.000997, ry=-175.461324, rz=20.570984, shoulder=lefty, elbow=epositive, wrist=wpositive, fatherId=frmaster[0]}
  [158] = {x=-70.188012, y=-2.561577, z=116.358122, rx=0.000228, ry=-175.460862, rz=20.571116, shoulder=lefty, elbow=epositive, wrist=wpositive, fatherId=frmaster[0]}
  [159] = {x=-70.181597, y=-2.561146, z=111.359101, rx=-0.00036, ry=-175.460979, rz=20.571392, shoulder=lefty, elbow=epositive, wrist=wpositive, fatherId=frmaster[0]}
  [160] = {x=-70.186856, y=-2.562635, z=101.36022, rx=0.000049, ry=-175.46102, rz=20.571062, shoulder=lefty, elbow=epositive, wrist=wpositive, fatherId=frmaster[0]}
  [161] = {x=-65.655471, y=-4.488719, z=104.643099, rx=-0.000151, ry=-172.679256, rz=18.950277, shoulder=lefty, elbow=epositive, wrist=wpositive, fatherId=frmaster[0]}
  [162] = {x=-62.242142, y=-5.688169, z=106.820543, rx=-0.000222, ry=-170.71867, rz=17.976729, shoulder=lefty, elbow=epositive, wrist=wpositive, fatherId=frmaster[0]}
  [163] = {x=-57.90117, y=-6.989821, z=109.313429, rx=-0.000644, ry=-168.324507, rz=16.936516, shoulder=lefty, elbow=epositive, wrist=wpositive, fatherId=frmaster[0]}
  [164] = {x=-55.30165, y=-7.668076, z=110.668104, rx=-0.00133, ry=-166.93388, rz=16.40052, shoulder=lefty, elbow=epositive, wrist=wpositive, fatherId=frmaster[0]}
  [165] = {x=-52.221943, y=-8.407272, z=112.170504, rx=-0.000258, ry=-165.315233, rz=15.819279, shoulder=lefty, elbow=epositive, wrist=wpositive, fatherId=frmaster[0]}
  [166] = {x=-48.656768, y=-9.171728, z=113.763691, rx=-0.00026, ry=-163.480402, rz=15.225259, shoulder=lefty, elbow=epositive, wrist=wpositive, fatherId=frmaster[0]}
  [167] = {x=-44.535561, y=-9.95158, z=115.419029, rx=-0.000976, ry=-161.400137, rz=14.618473, shoulder=lefty, elbow=epositive, wrist=wpositive, fatherId=frmaster[0]}
  [168] = {x=-39.894192, y=-10.715702, z=117.089206, rx=-0.000967, ry=-159.090682, rz=14.028421, shoulder=lefty, elbow=epositive, wrist=wpositive, fatherId=frmaster[0]}
  [169] = {x=-34.666317, y=-11.468884, z=118.713677, rx=-0.000844, ry=-156.530981, rz=13.444845, shoulder=lefty, elbow=epositive, wrist=wpositive, fatherId=frmaster[0]}
  [170] = {x=-28.887336, y=-12.184274, z=120.216655, rx=-0.000328, ry=-153.740419, rz=12.892649, shoulder=lefty, elbow=epositive, wrist=wpositive, fatherId=frmaster[0]}
  [171] = {x=-25.792943, y=-12.533702, z=120.889846, rx=-0.001232, ry=-152.260764, rz=12.623335, shoulder=lefty, elbow=epositive, wrist=wpositive, fatherId=frmaster[0]}
  [172] = {x=-22.564908, y=-12.873716, z=121.511598, rx=-0.001252, ry=-150.727048, rz=12.36006, shoulder=lefty, elbow=epositive, wrist=wpositive, fatherId=frmaster[0]}
  [173] = {x=-19.186652, y=-13.201047, z=122.068424, rx=-0.001327, ry=-149.126118, rz=12.108361, shoulder=lefty, elbow=epositive, wrist=wpositive, fatherId=frmaster[0]}
  [174] = {x=-15.643629, y=-13.520541, z=122.546216, rx=0.000126, ry=-147.457536, rz=11.860567, shoulder=lefty, elbow=epositive, wrist=wpositive, fatherId=frmaster[0]}
  [175] = {x=-11.939599, y=-13.838982, z=122.93158, rx=-0.000025, ry=-145.719372, rz=11.616135, shoulder=lefty, elbow=epositive, wrist=wpositive, fatherId=frmaster[0]}
  [176] = {x=-8.076918, y=-14.152946, z=123.211578, rx=-0.000823, ry=-143.9108, rz=11.374381, shoulder=lefty, elbow=epositive, wrist=wpositive, fatherId=frmaster[0]}
  [177] = {x=-4.053293, y=-14.451269, z=123.378323, rx=-0.000369, ry=-142.026575, rz=11.144782, shoulder=lefty, elbow=epositive, wrist=wpositive, fatherId=frmaster[0]}
  [178] = {x=-0.074753, y=-14.737841, z=123.404145, rx=-0.00165, ry=-140.16442, rz=10.924938, shoulder=lefty, elbow=epositive, wrist=wpositive, fatherId=frmaster[0]}
  [179] = {x=3.852205, y=-15.005731, z=123.313318, rx=-0.000892, ry=-138.326027, rz=10.715912, shoulder=lefty, elbow=epositive, wrist=wpositive, fatherId=frmaster[0]}
  [180] = {x=7.716616, y=-15.264764, z=123.093226, rx=-0.001219, ry=-136.513961, rz=10.515303, shoulder=lefty, elbow=epositive, wrist=wpositive, fatherId=frmaster[0]}
  [181] = {x=6.023663, y=-12.459759, z=123.553205, rx=-0.000508, ry=-137.110497, rz=12.853188, shoulder=lefty, elbow=epositive, wrist=wpositive, fatherId=frmaster[0]}
  [182] = {x=5.042073, y=-9.242716, z=123.915552, rx=-0.001829, ry=-137.391694, rz=15.473786, shoulder=lefty, elbow=epositive, wrist=wpositive, fatherId=frmaster[0]}
  [183] = {x=5.444959, y=-5.62198, z=124.138646, rx=-0.001624, ry=-137.06603, rz=18.36147, shoulder=lefty, elbow=epositive, wrist=wpositive, fatherId=frmaster[0]}
  [184] = {x=6.806434, y=-1.604055, z=124.197825, rx=-0.001709, ry=-136.346358, rz=21.519622, shoulder=lefty, elbow=epositive, wrist=wpositive, fatherId=frmaster[0]}
  [185] = {x=8.935655, y=2.5292, z=124.04304, rx=-0.00222, ry=-135.343654, rz=24.753008, shoulder=lefty, elbow=epositive, wrist=wpositive, fatherId=frmaster[0]}
  [186] = {x=12.034555, y=6.646495, z=123.609148, rx=-0.001789, ry=-133.954741, rz=27.973235, shoulder=lefty, elbow=epositive, wrist=wpositive, fatherId=frmaster[0]}
  [187] = {x=15.064777, y=10.744597, z=122.943806, rx=-0.002998, ry=-132.666375, rz=31.194437, shoulder=lefty, elbow=epositive, wrist=wpositive, fatherId=frmaster[0]}
  [188] = {x=18.862609, y=14.810745, z=121.94017, rx=-0.00319, ry=-131.071443, rz=34.411201, shoulder=lefty, elbow=epositive, wrist=wpositive, fatherId=frmaster[0]}
  [189] = {x=21.810028, y=18.953484, z=120.802874, rx=-0.001691, ry=-129.947568, rz=37.717936, shoulder=lefty, elbow=epositive, wrist=wpositive, fatherId=frmaster[0]}
  [190] = {x=25.289765, y=22.946049, z=119.329127, rx=-0.00265, ry=-128.601658, rz=40.957943, shoulder=lefty, elbow=epositive, wrist=wpositive, fatherId=frmaster[0]}
  [191] = {x=27.54309, y=26.880776, z=117.898839, rx=-0.001307, ry=-127.90927, rz=44.211596, shoulder=lefty, elbow=epositive, wrist=wpositive, fatherId=frmaster[0]}
  [192] = {x=30.26726, y=30.607326, z=116.187326, rx=-0.002618, ry=-127.011613, rz=47.366834, shoulder=lefty, elbow=epositive, wrist=wpositive, fatherId=frmaster[0]}
  [193] = {x=32.494978, y=34.218432, z=114.427543, rx=-0.003048, ry=-126.397593, rz=50.503731, shoulder=lefty, elbow=epositive, wrist=wpositive, fatherId=frmaster[0]}
  [194] = {x=35.113749, y=37.657955, z=112.409445, rx=-0.001693, ry=-125.609423, rz=53.579091, shoulder=lefty, elbow=epositive, wrist=wpositive, fatherId=frmaster[0]}
  [195] = {x=38.043252, y=40.883302, z=110.124593, rx=-0.002981, ry=-124.662527, rz=56.562689, shoulder=lefty, elbow=epositive, wrist=wpositive, fatherId=frmaster[0]}
  [196] = {x=41.123477, y=43.876486, z=107.647896, rx=-0.00208, ry=-123.613287, rz=59.433069, shoulder=lefty, elbow=epositive, wrist=wpositive, fatherId=frmaster[0]}
  [197] = {x=44.929669, y=46.507611, z=104.753884, rx=-0.003225, ry=-122.096717, rz=62.068846, shoulder=lefty, elbow=epositive, wrist=wpositive, fatherId=frmaster[0]}
  [198] = {x=48.653011, y=48.986114, z=101.682869, rx=-0.002256, ry=-120.5697, rz=64.64408, shoulder=lefty, elbow=epositive, wrist=wpositive, fatherId=frmaster[0]}
  [199] = {x=51.05339, y=50.032365, z=99.823902, rx=-0.003927, ry=-119.421725, rz=65.77687, shoulder=lefty, elbow=epositive, wrist=wpositive, fatherId=frmaster[0]}
  [200] = {x=53.791156, y=51.04185, z=97.71372, rx=-0.004642, ry=-118.046544, rz=66.88713, shoulder=lefty, elbow=epositive, wrist=wpositive, fatherId=frmaster[0]}
  [201] = {x=56.953868, y=52.016874, z=95.220966, rx=-0.003685, ry=-116.374614, rz=67.983851, shoulder=lefty, elbow=epositive, wrist=wpositive, fatherId=frmaster[0]}
  [202] = {x=60.5108, y=52.963909, z=92.301263, rx=-0.001568, ry=-114.401878, rz=69.069983, shoulder=lefty, elbow=epositive, wrist=wpositive, fatherId=frmaster[0]}
  [203] = {x=57.890367, y=52.941937, z=94.034918, rx=-0.003051, ry=-116.050047, rz=69.025533, shoulder=lefty, elbow=epositive, wrist=wpositive, fatherId=frmaster[0]}
  [204] = {x=55.459565, y=52.924385, z=95.558004, rx=-0.003596, ry=-117.555505, rz=68.983435, shoulder=lefty, elbow=epositive, wrist=wpositive, fatherId=frmaster[0]}
  [205] = {x=51.294271, y=52.89043, z=97.996514, rx=-0.001257, ry=-120.089167, rz=68.897689, shoulder=lefty, elbow=epositive, wrist=wpositive, fatherId=frmaster[0]}
  [206] = {x=47.775731, y=52.837382, z=99.887079, rx=-0.002, ry=-122.188827, rz=68.794993, shoulder=lefty, elbow=epositive, wrist=wpositive, fatherId=frmaster[0]}
  [207] = {x=43.99782, y=52.774725, z=101.739703, rx=-0.002744, ry=-124.388318, rz=68.682576, shoulder=lefty, elbow=epositive, wrist=wpositive, fatherId=frmaster[0]}
  [208] = {x=39.981614, y=52.619197, z=103.552994, rx=-0.003696, ry=-126.649809, rz=68.468492, shoulder=lefty, elbow=epositive, wrist=wpositive, fatherId=frmaster[0]}
  [209] = {x=35.789346, y=52.460485, z=105.253791, rx=-0.000589, ry=-128.969095, rz=68.252264, shoulder=lefty, elbow=epositive, wrist=wpositive, fatherId=frmaster[0]}
  [210] = {x=31.601795, y=52.284408, z=106.7468, rx=-0.001532, ry=-131.237279, rz=68.019263, shoulder=lefty, elbow=epositive, wrist=wpositive, fatherId=frmaster[0]}
  [211] = {x=27.438272, y=52.090828, z=108.050575, rx=-0.001868, ry=-133.456539, rz=67.769846, shoulder=lefty, elbow=epositive, wrist=wpositive, fatherId=frmaster[0]}
  [212] = {x=23.21378, y=51.812922, z=109.240942, rx=-0.002407, ry=-135.646933, rz=67.428001, shoulder=lefty, elbow=epositive, wrist=wpositive, fatherId=frmaster[0]}
  [213] = {x=18.743706, y=51.514645, z=110.304576, rx=-0.001429, ry=-137.933189, rz=67.070428, shoulder=lefty, elbow=epositive, wrist=wpositive, fatherId=frmaster[0]}
  [214] = {x=13.993428, y=51.19706, z=111.213118, rx=-0.001024, ry=-140.330662, rz=66.692984, shoulder=lefty, elbow=epositive, wrist=wpositive, fatherId=frmaster[0]}
  [215] = {x=9.124318, y=50.846962, z=111.919866, rx=-0.001423, ry=-142.763438, rz=66.286785, shoulder=lefty, elbow=epositive, wrist=wpositive, fatherId=frmaster[0]}
  [216] = {x=4.283267, y=50.411595, z=112.456612, rx=-0.001123, ry=-145.126518, rz=65.795998, shoulder=lefty, elbow=epositive, wrist=wpositive, fatherId=frmaster[0]}
  [217] = {x=-0.577211, y=49.922299, z=112.797447, rx=-0.001549, ry=-147.468866, rz=65.255497, shoulder=lefty, elbow=epositive, wrist=wpositive, fatherId=frmaster[0]}
  [218] = {x=-5.41872, y=49.372541, z=112.948393, rx=-0.000765, ry=-149.777785, rz=64.660093, shoulder=lefty, elbow=epositive, wrist=wpositive, fatherId=frmaster[0]}
  [219] = {x=-10.213936, y=48.748615, z=112.913124, rx=-0.000445, ry=-152.029949, rz=63.999234, shoulder=lefty, elbow=epositive, wrist=wpositive, fatherId=frmaster[0]}
  [220] = {x=-14.884154, y=48.042138, z=112.715994, rx=-0.001291, ry=-154.190388, rz=63.26674, shoulder=lefty, elbow=epositive, wrist=wpositive, fatherId=frmaster[0]}
  [221] = {x=-19.447226, y=47.239031, z=112.380346, rx=-0.000761, ry=-156.268251, rz=62.451755, shoulder=lefty, elbow=epositive, wrist=wpositive, fatherId=frmaster[0]}
  [222] = {x=-23.855402, y=46.328388, z=111.923012, rx=-0.000024, ry=-158.242856, rz=61.541728, shoulder=lefty, elbow=epositive, wrist=wpositive, fatherId=frmaster[0]}
  [223] = {x=-28.094929, y=45.28744, z=111.366501, rx=-0.001113, ry=-160.096268, rz=60.525998, shoulder=lefty, elbow=epositive, wrist=wpositive, fatherId=frmaster[0]}
  [224] = {x=-32.155226, y=44.135835, z=110.739017, rx=0.00011, ry=-161.837413, rz=59.420297, shoulder=lefty, elbow=epositive, wrist=wpositive, fatherId=frmaster[0]}
  [225] = {x=-35.970547, y=42.902831, z=110.040463, rx=-0.000981, ry=-163.447146, rz=58.254377, shoulder=lefty, elbow=epositive, wrist=wpositive, fatherId=frmaster[0]}
  [226] = {x=-42.880302, y=40.212603, z=108.556292, rx=-0.000316, ry=-166.292077, rz=55.764728, shoulder=lefty, elbow=epositive, wrist=wpositive, fatherId=frmaster[0]}
  [227] = {x=-49.024244, y=37.201229, z=106.989523, rx=-0.001168, ry=-168.736881, rz=53.054563, shoulder=lefty, elbow=epositive, wrist=wpositive, fatherId=frmaster[0]}
  [228] = {x=-54.340997, y=33.858737, z=105.473898, rx=-0.001202, ry=-170.773593, rz=50.121392, shoulder=lefty, elbow=epositive, wrist=wpositive, fatherId=frmaster[0]}
  [229] = {x=-59.016727, y=30.102997, z=104.037178, rx=-0.000911, ry=-172.486442, rz=46.913888, shoulder=lefty, elbow=epositive, wrist=wpositive, fatherId=frmaster[0]}
  [230] = {x=-63.006363, y=25.804715, z=102.783723, rx=-0.000944, ry=-173.859315, rz=43.334617, shoulder=lefty, elbow=epositive, wrist=wpositive, fatherId=frmaster[0]}
  [231] = {x=-69.147803, y=15.172479, z=100.801054, rx=-0.000301, ry=-175.823411, rz=34.802868, shoulder=lefty, elbow=epositive, wrist=wpositive, fatherId=frmaster[0]}
  [232] = {x=-72.314741, y=5.296055, z=99.404785, rx=0.000497, ry=-177.026794, rz=27.000477, shoulder=lefty, elbow=epositive, wrist=wpositive, fatherId=frmaster[0]}
  [233] = {x=-72.319472, y=5.293472, z=109.398913, rx=-0.00012, ry=-177.027506, rz=26.998905, shoulder=lefty, elbow=epositive, wrist=wpositive, fatherId=frmaster[0]}
  [234] = {x=-72.317875, y=5.291508, z=114.399852, rx=-0.000462, ry=-177.027584, rz=26.999126, shoulder=lefty, elbow=epositive, wrist=wpositive, fatherId=frmaster[0]}
  [235] = {x=-71.828243, y=5.29286, z=123.893616, rx=0.000101, ry=-177.027112, rz=26.99867, shoulder=lefty, elbow=epositive, wrist=wpositive, fatherId=frmaster[0]}
  [236] = {x=-71.650279, y=5.202066, z=123.884373, rx=-179.999899, ry=-2.972888, rz=26.99867, shoulder=lefty, elbow=epositive, wrist=wpositive, fatherId=frmaster[0]}
  [237] = {x=-72.139912, y=5.200713, z=114.390612, rx=179.999538, ry=-2.972416, rz=26.999126, shoulder=lefty, elbow=epositive, wrist=wpositive, fatherId=frmaster[0]}
  [238] = {x=-72.141509, y=5.202677, z=109.389672, rx=179.99988, ry=-2.972494, rz=26.998905, shoulder=lefty, elbow=epositive, wrist=wpositive, fatherId=frmaster[0]}
  [239] = {x=-72.136781, y=5.205256, z=99.395541, rx=-179.999503, ry=-2.973206, rz=27.000477, shoulder=lefty, elbow=epositive, wrist=wpositive, fatherId=frmaster[0]}
  [240] = {x=-68.984015, y=15.058328, z=100.789094, rx=179.999699, ry=-4.176589, rz=34.802868, shoulder=lefty, elbow=epositive, wrist=wpositive, fatherId=frmaster[0]}
  [241] = {x=-62.861726, y=25.667463, z=102.768164, rx=179.999056, ry=-6.140685, rz=43.334617, shoulder=lefty, elbow=epositive, wrist=wpositive, fatherId=frmaster[0]}
  [242] = {x=-58.88128, y=29.956932, z=104.019316, rx=179.999089, ry=-7.513558, rz=46.913888, shoulder=lefty, elbow=epositive, wrist=wpositive, fatherId=frmaster[0]}
  [243] = {x=-54.214424, y=33.705256, z=105.453341, rx=179.998798, ry=-9.226407, rz=50.121392, shoulder=lefty, elbow=epositive, wrist=wpositive, fatherId=frmaster[0]}
  [244] = {x=-48.906348, y=37.041387, z=106.966048, rx=179.998832, ry=-11.263119, rz=53.054563, shoulder=lefty, elbow=epositive, wrist=wpositive, fatherId=frmaster[0]}
  [245] = {x=-42.770988, y=40.047256, z=108.529629, rx=179.999684, ry=-13.707923, rz=55.764728, shoulder=lefty, elbow=epositive, wrist=wpositive, fatherId=frmaster[0]}
  [246] = {x=-35.869678, y=42.732752, z=110.010486, rx=179.999019, ry=-16.552854, rz=58.254377, shoulder=lefty, elbow=epositive, wrist=wpositive, fatherId=frmaster[0]}
  [247] = {x=-32.058548, y=43.963651, z=110.707301, rx=-179.99989, ry=-18.162587, rz=59.420297, shoulder=lefty, elbow=epositive, wrist=wpositive, fatherId=frmaster[0]}
  [248] = {x=-28.002402, y=45.113323, z=111.333003, rx=179.998887, ry=-19.903732, rz=60.525998, shoulder=lefty, elbow=epositive, wrist=wpositive, fatherId=frmaster[0]}
  [249] = {x=-23.766887, y=46.152555, z=111.887685, rx=179.999976, ry=-21.757144, rz=61.541728, shoulder=lefty, elbow=epositive, wrist=wpositive, fatherId=frmaster[0]}
  [250] = {x=-19.362549, y=47.061707, z=112.343122, rx=179.999239, ry=-23.731749, rz=62.451755, shoulder=lefty, elbow=epositive, wrist=wpositive, fatherId=frmaster[0]}
  [251] = {x=-14.803161, y=47.863515, z=112.676828, rx=179.998709, ry=-25.809612, rz=63.26674, shoulder=lefty, elbow=epositive, wrist=wpositive, fatherId=frmaster[0]}
  [252] = {x=-10.1365, y=48.568857, z=112.872005, rx=179.999555, ry=-27.970051, rz=63.999234, shoulder=lefty, elbow=epositive, wrist=wpositive, fatherId=frmaster[0]}
  [253] = {x=-5.344757, y=49.191783, z=112.90531, rx=179.999235, ry=-30.222215, rz=64.660093, shoulder=lefty, elbow=epositive, wrist=wpositive, fatherId=frmaster[0]}
  [254] = {x=-0.506631, y=49.740661, z=112.752434, rx=179.998451, ry=-32.531134, rz=65.255497, shoulder=lefty, elbow=epositive, wrist=wpositive, fatherId=frmaster[0]}
  [255] = {x=4.350539, y=50.229176, z=112.409732, rx=179.998877, ry=-34.873482, rz=65.795998, shoulder=lefty, elbow=epositive, wrist=wpositive, fatherId=frmaster[0]}
  [256] = {x=9.188354, y=50.663847, z=111.8712, rx=179.998577, ry=-37.236562, rz=66.286785, shoulder=lefty, elbow=epositive, wrist=wpositive, fatherId=frmaster[0]}
  [257] = {x=14.054339, y=51.01338, z=111.162607, rx=179.998976, ry=-39.669338, rz=66.692984, shoulder=lefty, elbow=epositive, wrist=wpositive, fatherId=frmaster[0]}
  [258] = {x=18.801551, y=51.330447, z=110.252374, rx=179.998571, ry=-42.066811, rz=67.070428, shoulder=lefty, elbow=epositive, wrist=wpositive, fatherId=frmaster[0]}
  [259] = {x=23.268674, y=51.62824, z=109.187283, rx=179.997593, ry=-44.353067, rz=67.428001, shoulder=lefty, elbow=epositive, wrist=wpositive, fatherId=frmaster[0]}
  [260] = {x=27.490315, y=51.905692, z=107.995656, rx=179.998132, ry=-46.543461, rz=67.769846, shoulder=lefty, elbow=epositive, wrist=wpositive, fatherId=frmaster[0]}
  [261] = {x=31.651141, y=52.098945, z=106.690512, rx=179.998468, ry=-48.762721, rz=68.019263, shoulder=lefty, elbow=epositive, wrist=wpositive, fatherId=frmaster[0]}
  [262] = {x=35.835951, y=52.27472, z=105.196178, rx=179.999411, ry=-51.030905, rz=68.252264, shoulder=lefty, elbow=epositive, wrist=wpositive, fatherId=frmaster[0]}
  [263] = {x=40.02543, y=52.43315, z=103.494115, rx=179.996304, ry=-53.350191, rz=68.468492, shoulder=lefty, elbow=epositive, wrist=wpositive, fatherId=frmaster[0]}
  [264] = {x=44.038885, y=52.588406, z=101.679712, rx=179.997256, ry=-55.611682, rz=68.682576, shoulder=lefty, elbow=epositive, wrist=wpositive, fatherId=frmaster[0]}
  [265] = {x=47.814268, y=52.650921, z=99.825864, rx=179.998, ry=-57.811173, rz=68.794993, shoulder=lefty, elbow=epositive, wrist=wpositive, fatherId=frmaster[0]}
  [266] = {x=51.330371, y=52.703841, z=97.934214, rx=179.998743, ry=-59.910833, rz=68.897689, shoulder=lefty, elbow=epositive, wrist=wpositive, fatherId=frmaster[0]}
  [267] = {x=55.492747, y=52.737685, z=95.494425, rx=179.996404, ry=-62.444495, rz=68.983435, shoulder=lefty, elbow=epositive, wrist=wpositive, fatherId=frmaster[0]}
  [268] = {x=57.921806, y=52.755186, z=93.970611, rx=179.996949, ry=-63.949953, rz=69.025533, shoulder=lefty, elbow=epositive, wrist=wpositive, fatherId=frmaster[0]}
  [269] = {x=60.540316, y=52.777104, z=92.236205, rx=179.998432, ry=-65.598122, rz=69.069983, shoulder=lefty, elbow=epositive, wrist=wpositive, fatherId=frmaster[0]}
  [270] = {x=56.987174, y=51.831454, z=95.153808, rx=179.996315, ry=-63.625386, rz=67.983851, shoulder=lefty, elbow=epositive, wrist=wpositive, fatherId=frmaster[0]}
  [271] = {x=53.82807, y=50.857898, z=97.644446, rx=179.995358, ry=-61.953456, rz=66.88713, shoulder=lefty, elbow=epositive, wrist=wpositive, fatherId=frmaster[0]}
  [272] = {x=51.093699, y=49.849969, z=99.75244, rx=179.996073, ry=-60.578275, rz=65.77687, shoulder=lefty, elbow=epositive, wrist=wpositive, fatherId=frmaster[0]}
  [273] = {x=48.69657, y=48.805378, z=101.609133, rx=179.997744, ry=-59.4303, rz=64.64408, shoulder=lefty, elbow=epositive, wrist=wpositive, fatherId=frmaster[0]}
  [274] = {x=44.979447, y=46.330905, z=104.674531, rx=179.996775, ry=-57.903283, rz=62.068846, shoulder=lefty, elbow=epositive, wrist=wpositive, fatherId=frmaster[0]}
  [275] = {x=41.179782, y=43.704276, z=107.5632, rx=179.99792, ry=-56.386713, rz=59.433069, shoulder=lefty, elbow=epositive, wrist=wpositive, fatherId=frmaster[0]}
  [276] = {x=38.10593, y=40.716399, z=110.033956, rx=179.997019, ry=-55.337473, rz=56.562689, shoulder=lefty, elbow=epositive, wrist=wpositive, fatherId=frmaster[0]}
  [277] = {x=35.182888, y=37.497017, z=112.312911, rx=179.998307, ry=-54.390577, rz=53.579091, shoulder=lefty, elbow=epositive, wrist=wpositive, fatherId=frmaster[0]}
  [278] = {x=32.57046, y=34.064094, z=114.325161, rx=179.996952, ry=-53.602407, rz=50.503731, shoulder=lefty, elbow=epositive, wrist=wpositive, fatherId=frmaster[0]}
  [279] = {x=30.348804, y=30.46018, z=116.079166, rx=179.997382, ry=-52.988387, rz=47.366834, shoulder=lefty, elbow=epositive, wrist=wpositive, fatherId=frmaster[0]}
  [280] = {x=27.631168, y=26.741312, z=117.785738, rx=179.998693, ry=-52.09073, rz=44.211596, shoulder=lefty, elbow=epositive, wrist=wpositive, fatherId=frmaster[0]}
  [281] = {x=25.383998, y=22.814943, z=119.211097, rx=179.99735, ry=-51.398342, rz=40.957943, shoulder=lefty, elbow=epositive, wrist=wpositive, fatherId=frmaster[0]}
  [282] = {x=21.91161, y=18.831126, z=120.681592, rx=179.998309, ry=-50.052432, rz=37.717936, shoulder=lefty, elbow=epositive, wrist=wpositive, fatherId=frmaster[0]}
  [283] = {x=18.971014, y=14.697712, z=121.815784, rx=179.99681, ry=-48.928557, rz=34.411201, shoulder=lefty, elbow=epositive, wrist=wpositive, fatherId=frmaster[0]}
  [284] = {x=15.180725, y=10.641001, z=122.818012, rx=179.997002, ry=-47.333625, rz=31.194437, shoulder=lefty, elbow=epositive, wrist=wpositive, fatherId=frmaster[0]}
  [285] = {x=12.157154, y=6.552679, z=123.481995, rx=179.998211, ry=-46.045259, rz=27.973235, shoulder=lefty, elbow=epositive, wrist=wpositive, fatherId=frmaster[0]}
  [286] = {x=9.064851, y=2.445453, z=123.915388, rx=179.99778, ry=-44.656346, rz=24.753008, shoulder=lefty, elbow=epositive, wrist=wpositive, fatherId=frmaster[0]}
  [287] = {x=6.941052, y=-1.677423, z=124.069391, rx=179.998291, ry=-43.653642, rz=21.519622, shoulder=lefty, elbow=epositive, wrist=wpositive, fatherId=frmaster[0]}
  [288] = {x=5.583931, y=-5.684986, z=124.009352, rx=179.998376, ry=-42.93397, rz=18.36147, shoulder=lefty, elbow=epositive, wrist=wpositive, fatherId=frmaster[0]}
  [289] = {x=5.183937, y=-9.29608, z=123.785065, rx=179.998171, ry=-42.608306, rz=15.473786, shoulder=lefty, elbow=epositive, wrist=wpositive, fatherId=frmaster[0]}
  [290] = {x=6.166525, y=-12.504251, z=123.420499, rx=179.999492, ry=-42.889503, rz=12.853188, shoulder=lefty, elbow=epositive, wrist=wpositive, fatherId=frmaster[0]}
  [291] = {x=7.859288, y=-15.301266, z=122.957903, rx=179.998781, ry=-43.486039, rz=10.515303, shoulder=lefty, elbow=epositive, wrist=wpositive, fatherId=frmaster[0]}
  [292] = {x=3.998988, y=-15.042921, z=123.182659, rx=179.999108, ry=-41.673973, rz=10.715912, shoulder=lefty, elbow=epositive, wrist=wpositive, fatherId=frmaster[0]}
  [293] = {x=0.076041, y=-14.775749, z=123.27835, rx=179.99835, ry=-39.83558, rz=10.924938, shoulder=lefty, elbow=epositive, wrist=wpositive, fatherId=frmaster[0]}
  [294] = {x=-3.898607, y=-14.489927, z=123.257585, rx=179.999631, ry=-37.973425, rz=11.144782, shoulder=lefty, elbow=epositive, wrist=wpositive, fatherId=frmaster[0]}
  [295] = {x=-7.918472, y=-14.192392, z=123.096083, rx=179.999177, ry=-36.0892, rz=11.374381, shoulder=lefty, elbow=epositive, wrist=wpositive, fatherId=frmaster[0]}
  [296] = {x=-11.777726, y=-13.879253, z=122.821238, rx=179.999975, ry=-34.280628, rz=11.616135, shoulder=lefty, elbow=epositive, wrist=wpositive, fatherId=frmaster[0]}
  [297] = {x=-15.47863, y=-13.561647, z=122.440928, rx=-179.999874, ry=-32.542464, rz=11.860567, shoulder=lefty, elbow=epositive, wrist=wpositive, fatherId=frmaster[0]}
  [298] = {x=-19.018811, y=-13.243002, z=121.968078, rx=179.998673, ry=-30.873882, rz=12.108361, shoulder=lefty, elbow=epositive, wrist=wpositive, fatherId=frmaster[0]}
  [299] = {x=-22.394492, y=-12.916529, z=121.416072, rx=179.998748, ry=-29.272952, rz=12.36006, shoulder=lefty, elbow=epositive, wrist=wpositive, fatherId=frmaster[0]}
  [300] = {x=-25.620207, y=-12.577412, z=120.799007, rx=179.998768, ry=-27.739236, rz=12.623335, shoulder=lefty, elbow=epositive, wrist=wpositive, fatherId=frmaster[0]}
  [301] = {x=-28.712498, y=-12.2289, z=120.130398, rx=179.999672, ry=-26.259581, rz=12.892649, shoulder=lefty, elbow=epositive, wrist=wpositive, fatherId=frmaster[0]}
  [302] = {x=-34.48789, y=-11.515387, z=118.63621, rx=179.999156, ry=-23.469019, rz=13.444845, shoulder=lefty, elbow=epositive, wrist=wpositive, fatherId=frmaster[0]}
  [303] = {x=-39.712935, y=-10.764184, z=117.019957, rx=179.999033, ry=-20.909318, rz=14.028421, shoulder=lefty, elbow=epositive, wrist=wpositive, fatherId=frmaster[0]}
  [304] = {x=-44.352144, y=-10.002058, z=115.357303, rx=179.999024, ry=-18.599863, rz=14.618473, shoulder=lefty, elbow=epositive, wrist=wpositive, fatherId=frmaster[0]}
  [305] = {x=-48.471753, y=-9.224252, z=113.708819, rx=179.99974, ry=-16.519598, rz=15.225259, shoulder=lefty, elbow=epositive, wrist=wpositive, fatherId=frmaster[0]}
  [306] = {x=-52.035803, y=-8.461793, z=112.121724, rx=179.999742, ry=-14.684767, rz=15.819279, shoulder=lefty, elbow=epositive, wrist=wpositive, fatherId=frmaster[0]}
  [307] = {x=-55.114755, y=-7.724547, z=110.62473, rx=179.99867, ry=-13.06612, rz=16.40052, shoulder=lefty, elbow=epositive, wrist=wpositive, fatherId=frmaster[0]}
  [308] = {x=-57.713803, y=-7.048084, z=109.274711, rx=179.999356, ry=-11.675493, rz=16.936516, shoulder=lefty, elbow=epositive, wrist=wpositive, fatherId=frmaster[0]}
  [309] = {x=-62.054396, y=-5.749895, z=106.789862, rx=179.999778, ry=-9.28133, rz=17.976729, shoulder=lefty, elbow=epositive, wrist=wpositive, fatherId=frmaster[0]}
  [310] = {x=-65.467853, y=-4.553669, z=104.618996, rx=179.999849, ry=-7.320744, rz=18.950277, shoulder=lefty, elbow=epositive, wrist=wpositive, fatherId=frmaster[0]}
  [311] = {x=-70.000196, y=-2.632909, z=101.345402, rx=-179.999951, ry=-4.53898, rz=20.571062, shoulder=lefty, elbow=epositive, wrist=wpositive, fatherId=frmaster[0]}
  [312] = {x=-69.994937, y=-2.631421, z=111.344283, rx=179.99964, ry=-4.539021, rz=20.571392, shoulder=lefty, elbow=epositive, wrist=wpositive, fatherId=frmaster[0]}
  [313] = {x=-70.001351, y=-2.631851, z=116.343303, rx=-179.999772, ry=-4.539138, rz=20.571116, shoulder=lefty, elbow=epositive, wrist=wpositive, fatherId=frmaster[0]}
  [314] = {x=-66.075805, y=-2.426028, z=114.78733, rx=179.842158, ry=-7.534906, rz=20.567234, shoulder=lefty, elbow=epositive, wrist=wpositive, fatherId=frmaster[0]}
  [315] = {x=-65.82094, y=-2.412764, z=119.779835, rx=179.84275, ry=-7.535023, rz=20.566988, shoulder=lefty, elbow=epositive, wrist=wpositive, fatherId=frmaster[0]}
  [316] = {fatherId=frmaster[0]}
  [317] = {fatherId=frmaster[0]}
  [318] = {fatherId=frmaster[0]}
  [319] = {fatherId=frmaster[0]}
  [320] = {fatherId=frmaster[0]}
  [321] = {fatherId=frmaster[0]}
  [322] = {fatherId=frmaster[0]}
  [323] = {fatherId=frmaster[0]}
  [324] = {fatherId=frmaster[0]}
  [325] = {fatherId=frmaster[0]}
  [326] = {fatherId=frmaster[0]}
  [327] = {fatherId=frmaster[0]}
  [328] = {fatherId=frmaster[0]}
  [329] = {fatherId=frmaster[0]}
  [330] = {fatherId=frmaster[0]}
  [331] = {fatherId=frmaster[0]}
  [332] = {fatherId=frmaster[0]}
  [333] = {fatherId=frmaster[0]}
  [334] = {fatherId=frmaster[0]}
  [335] = {fatherId=frmaster[0]}
  [336] = {fatherId=frmaster[0]}
  [337] = {fatherId=frmaster[0]}
  [338] = {fatherId=frmaster[0]}
  [339] = {fatherId=frmaster[0]}
  [340] = {fatherId=frmaster[0]}
  [341] = {fatherId=frmaster[0]}
  [342] = {fatherId=frmaster[0]}
  [343] = {fatherId=frmaster[0]}
  [344] = {fatherId=frmaster[0]}
  [345] = {fatherId=frmaster[0]}
  [346] = {fatherId=frmaster[0]}
  [347] = {fatherId=frmaster[0]}
  [348] = {fatherId=frmaster[0]}
  [349] = {fatherId=frmaster[0]}
  [350] = {fatherId=frmaster[0]}
  [351] = {fatherId=frmaster[0]}
  [352] = {fatherId=frmaster[0]}
  [353] = {fatherId=frmaster[0]}
  [354] = {fatherId=frmaster[0]}
  [355] = {fatherId=frmaster[0]}
  [356] = {fatherId=frmaster[0]}
  [357] = {fatherId=frmaster[0]}
  [358] = {fatherId=frmaster[0]}
  [359] = {fatherId=frmaster[0]}
  [360] = {fatherId=frmaster[0]}
  [361] = {fatherId=frmaster[0]}
  [362] = {fatherId=frmaster[0]}
  [363] = {fatherId=frmaster[0]}
  [364] = {fatherId=frmaster[0]}
  [365] = {fatherId=frmaster[0]}
  [366] = {fatherId=frmaster[0]}
  [367] = {fatherId=frmaster[0]}
  [368] = {fatherId=frmaster[0]}
  [369] = {fatherId=frmaster[0]}
  [370] = {fatherId=frmaster[0]}
  [371] = {fatherId=frmaster[0]}
  [372] = {fatherId=frmaster[0]}
  [373] = {fatherId=frmaster[0]}
  [374] = {fatherId=frmaster[0]}
  [375] = {fatherId=frmaster[0]}
  [376] = {fatherId=frmaster[0]}
  [377] = {fatherId=frmaster[0]}
  [378] = {fatherId=frmaster[0]}
  [379] = {fatherId=frmaster[0]}
  [380] = {fatherId=frmaster[0]}
  [381] = {fatherId=frmaster[0]}
  [382] = {fatherId=frmaster[0]}
  [383] = {fatherId=frmaster[0]}
  [384] = {fatherId=frmaster[0]}
  [385] = {fatherId=frmaster[0]}
  [386] = {fatherId=frmaster[0]}
  [387] = {fatherId=frmaster[0]}
  [388] = {fatherId=frmaster[0]}
  [389] = {fatherId=frmaster[0]}
  [390] = {fatherId=frmaster[0]}
  [391] = {fatherId=frmaster[0]}
  [392] = {fatherId=frmaster[0]}
  [393] = {fatherId=frmaster[0]}
  [394] = {fatherId=frmaster[0]}
  [395] = {fatherId=frmaster[0]}
  [396] = {fatherId=frmaster[0]}
  [397] = {fatherId=frmaster[0]}
  [398] = {fatherId=frmaster[0]}
  [399] = {fatherId=frmaster[0]}
  [400] = {fatherId=frmaster[0]}
  [401] = {fatherId=frmaster[0]}
  [402] = {fatherId=frmaster[0]}
  [403] = {fatherId=frmaster[0]}
  [404] = {fatherId=frmaster[0]}
  [405] = {fatherId=frmaster[0]}
  [406] = {fatherId=frmaster[0]}
  [407] = {fatherId=frmaster[0]}
  [408] = {fatherId=frmaster[0]}
  [409] = {fatherId=frmaster[0]}
  [410] = {fatherId=frmaster[0]}
  [411] = {fatherId=frmaster[0]}
  [412] = {fatherId=frmaster[0]}
  [413] = {fatherId=frmaster[0]}
  [414] = {fatherId=frmaster[0]}
  [415] = {fatherId=frmaster[0]}
  [416] = {fatherId=frmaster[0]}
  [417] = {fatherId=frmaster[0]}
  [418] = {fatherId=frmaster[0]}
  [419] = {fatherId=frmaster[0]}
  [420] = {fatherId=frmaster[0]}
  [421] = {fatherId=frmaster[0]}
  [422] = {fatherId=frmaster[0]}
  [423] = {fatherId=frmaster[0]}
  [424] = {fatherId=frmaster[0]}
  [425] = {fatherId=frmaster[0]}
  [426] = {fatherId=frmaster[0]}
  [427] = {fatherId=frmaster[0]}
  [428] = {fatherId=frmaster[0]}
  [429] = {fatherId=frmaster[0]}
  [430] = {fatherId=frmaster[0]}
  [431] = {fatherId=frmaster[0]}
  [432] = {fatherId=frmaster[0]}
  [433] = {fatherId=frmaster[0]}
  [434] = {fatherId=frmaster[0]}
  [435] = {fatherId=frmaster[0]}
  [436] = {fatherId=frmaster[0]}
  [437] = {fatherId=frmaster[0]}
  [438] = {fatherId=frmaster[0]}
  [439] = {fatherId=frmaster[0]}
  [440] = {fatherId=frmaster[0]}
  [441] = {fatherId=frmaster[0]}
  [442] = {fatherId=frmaster[0]}
  [443] = {fatherId=frmaster[0]}
  [444] = {fatherId=frmaster[0]}
  [445] = {fatherId=frmaster[0]}
  [446] = {fatherId=frmaster[0]}
  [447] = {fatherId=frmaster[0]}
  [448] = {fatherId=frmaster[0]}
  [449] = {fatherId=frmaster[0]}
  [450] = {fatherId=frmaster[0]}
  [451] = {fatherId=frmaster[0]}
  [452] = {fatherId=frmaster[0]}
  [453] = {fatherId=frmaster[0]}
  [454] = {fatherId=frmaster[0]}
  [455] = {fatherId=frmaster[0]}
  [456] = {fatherId=frmaster[0]}
  [457] = {fatherId=frmaster[0]}
  [458] = {fatherId=frmaster[0]}
  [459] = {fatherId=frmaster[0]}
  [460] = {fatherId=frmaster[0]}
  [461] = {fatherId=frmaster[0]}
  [462] = {fatherId=frmaster[0]}
  [463] = {fatherId=frmaster[0]}
  [464] = {fatherId=frmaster[0]}
  [465] = {fatherId=frmaster[0]}
  [466] = {fatherId=frmaster[0]}
  [467] = {fatherId=frmaster[0]}
  [468] = {fatherId=frmaster[0]}
  [469] = {fatherId=frmaster[0]}
  [470] = {fatherId=frmaster[0]}
  [471] = {fatherId=frmaster[0]}
  [472] = {fatherId=frmaster[0]}
  [473] = {fatherId=frmaster[0]}
  [474] = {fatherId=frmaster[0]}
  [475] = {fatherId=frmaster[0]}
  [476] = {fatherId=frmaster[0]}
  [477] = {fatherId=frmaster[0]}
  [478] = {fatherId=frmaster[0]}
  [479] = {fatherId=frmaster[0]}
  [480] = {fatherId=frmaster[0]}
  [481] = {fatherId=frmaster[0]}
  [482] = {fatherId=frmaster[0]}
  [483] = {fatherId=frmaster[0]}
  [484] = {fatherId=frmaster[0]}
  [485] = {fatherId=frmaster[0]}
  [486] = {fatherId=frmaster[0]}
  [487] = {fatherId=frmaster[0]}
  [488] = {fatherId=frmaster[0]}
  [489] = {fatherId=frmaster[0]}
  [490] = {fatherId=frmaster[0]}
  [491] = {fatherId=frmaster[0]}
  [492] = {fatherId=frmaster[0]}
  [493] = {fatherId=frmaster[0]}
  [494] = {fatherId=frmaster[0]}
  [495] = {fatherId=frmaster[0]}
  [496] = {fatherId=frmaster[0]}
  [497] = {fatherId=frmaster[0]}
  [498] = {fatherId=frmaster[0]}
  [499] = {fatherId=frmaster[0]}
  [500] = {fatherId=frmaster[0]}
  [501] = {fatherId=frmaster[0]}
  [502] = {fatherId=frmaster[0]}
  [503] = {fatherId=frmaster[0]}
  [504] = {fatherId=frmaster[0]}
  [505] = {fatherId=frmaster[0]}
  [506] = {fatherId=frmaster[0]}
  [507] = {fatherId=frmaster[0]}
  [508] = {fatherId=frmaster[0]}
  [509] = {fatherId=frmaster[0]}
  [510] = {fatherId=frmaster[0]}
  [511] = {fatherId=frmaster[0]}
  [512] = {fatherId=frmaster[0]}
  [513] = {fatherId=frmaster[0]}
  [514] = {fatherId=frmaster[0]}
  [515] = {fatherId=frmaster[0]}
  [516] = {fatherId=frmaster[0]}
  [517] = {fatherId=frmaster[0]}
  [518] = {fatherId=frmaster[0]}
  [519] = {fatherId=frmaster[0]}
  [520] = {fatherId=frmaster[0]}
  [521] = {fatherId=frmaster[0]}
  [522] = {fatherId=frmaster[0]}
  [523] = {fatherId=frmaster[0]}
  [524] = {fatherId=frmaster[0]}
  [525] = {fatherId=frmaster[0]}
  [526] = {fatherId=frmaster[0]}
  [527] = {fatherId=frmaster[0]}
  [528] = {fatherId=frmaster[0]}
  [529] = {fatherId=frmaster[0]}
  [530] = {fatherId=frmaster[0]}
  [531] = {fatherId=frmaster[0]}
  [532] = {fatherId=frmaster[0]}
  [533] = {fatherId=frmaster[0]}
  [534] = {fatherId=frmaster[0]}
  [535] = {fatherId=frmaster[0]}
  [536] = {fatherId=frmaster[0]}
  [537] = {fatherId=frmaster[0]}
  [538] = {fatherId=frmaster[0]}
  [539] = {fatherId=frmaster[0]}
  [540] = {fatherId=frmaster[0]}
  [541] = {fatherId=frmaster[0]}
  [542] = {fatherId=frmaster[0]}
  [543] = {fatherId=frmaster[0]}
  [544] = {fatherId=frmaster[0]}
  [545] = {fatherId=frmaster[0]}
  [546] = {fatherId=frmaster[0]}
  [547] = {fatherId=frmaster[0]}
  [548] = {fatherId=frmaster[0]}
  [549] = {fatherId=frmaster[0]}
  [550] = {fatherId=frmaster[0]}
  [551] = {fatherId=frmaster[0]}
  [552] = {fatherId=frmaster[0]}
  [553] = {fatherId=frmaster[0]}
  [554] = {fatherId=frmaster[0]}
  [555] = {fatherId=frmaster[0]}
  [556] = {fatherId=frmaster[0]}
  [557] = {fatherId=frmaster[0]}
  [558] = {fatherId=frmaster[0]}
  [559] = {fatherId=frmaster[0]}
  [560] = {fatherId=frmaster[0]}
  [561] = {fatherId=frmaster[0]}
  [562] = {fatherId=frmaster[0]}
  [563] = {fatherId=frmaster[0]}
  [564] = {fatherId=frmaster[0]}
  [565] = {fatherId=frmaster[0]}
  [566] = {fatherId=frmaster[0]}
  [567] = {fatherId=frmaster[0]}
  [568] = {fatherId=frmaster[0]}
  [569] = {fatherId=frmaster[0]}
  [570] = {fatherId=frmaster[0]}
  [571] = {fatherId=frmaster[0]}
  [572] = {fatherId=frmaster[0]}
  [573] = {fatherId=frmaster[0]}
  [574] = {fatherId=frmaster[0]}
  [575] = {fatherId=frmaster[0]}
  [576] = {fatherId=frmaster[0]}
  [577] = {fatherId=frmaster[0]}
  [578] = {fatherId=frmaster[0]}
  [579] = {fatherId=frmaster[0]}
  [580] = {fatherId=frmaster[0]}
  [581] = {fatherId=frmaster[0]}
  [582] = {fatherId=frmaster[0]}
  [583] = {fatherId=frmaster[0]}
  [584] = {fatherId=frmaster[0]}
  [585] = {fatherId=frmaster[0]}
  [586] = {fatherId=frmaster[0]}
  [587] = {fatherId=frmaster[0]}
  [588] = {fatherId=frmaster[0]}
  [589] = {fatherId=frmaster[0]}
  [590] = {fatherId=frmaster[0]}
  [591] = {fatherId=frmaster[0]}
  [592] = {fatherId=frmaster[0]}
  [593] = {fatherId=frmaster[0]}
  [594] = {fatherId=frmaster[0]}
  [595] = {fatherId=frmaster[0]}
  [596] = {fatherId=frmaster[0]}
  [597] = {fatherId=frmaster[0]}
  [598] = {fatherId=frmaster[0]}
  [599] = {fatherId=frmaster[0]}
  [600] = {fatherId=frmaster[0]}
  [601] = {fatherId=frmaster[0]}
  [602] = {fatherId=frmaster[0]}
  [603] = {fatherId=frmaster[0]}
  [604] = {fatherId=frmaster[0]}
  [605] = {fatherId=frmaster[0]}
  [606] = {fatherId=frmaster[0]}
  [607] = {fatherId=frmaster[0]}
  [608] = {fatherId=frmaster[0]}
  [609] = {fatherId=frmaster[0]}
  [610] = {fatherId=frmaster[0]}
  [611] = {fatherId=frmaster[0]}
  [612] = {fatherId=frmaster[0]}
  [613] = {fatherId=frmaster[0]}
  [614] = {fatherId=frmaster[0]}
  [615] = {fatherId=frmaster[0]}
  [616] = {fatherId=frmaster[0]}
  [617] = {fatherId=frmaster[0]}
  [618] = {fatherId=frmaster[0]}
  [619] = {fatherId=frmaster[0]}
  [620] = {fatherId=frmaster[0]}
  [621] = {fatherId=frmaster[0]}
  [622] = {fatherId=frmaster[0]}
  [623] = {fatherId=frmaster[0]}
  [624] = {fatherId=frmaster[0]}
  [625] = {fatherId=frmaster[0]}
  [626] = {fatherId=frmaster[0]}
  [627] = {fatherId=frmaster[0]}
  [628] = {fatherId=frmaster[0]}
  [629] = {fatherId=frmaster[0]}
  [630] = {fatherId=frmaster[0]}
  [631] = {fatherId=frmaster[0]}
  [632] = {fatherId=frmaster[0]}
  [633] = {fatherId=frmaster[0]}
  [634] = {fatherId=frmaster[0]}
  [635] = {fatherId=frmaster[0]}
  [636] = {fatherId=frmaster[0]}
  [637] = {fatherId=frmaster[0]}
  [638] = {fatherId=frmaster[0]}
  [639] = {fatherId=frmaster[0]}
  [640] = {fatherId=frmaster[0]}
  [641] = {fatherId=frmaster[0]}
  [642] = {fatherId=frmaster[0]}
  [643] = {fatherId=frmaster[0]}
  [644] = {fatherId=frmaster[0]}
  [645] = {fatherId=frmaster[0]}
  [646] = {fatherId=frmaster[0]}
  [647] = {fatherId=frmaster[0]}
  [648] = {fatherId=frmaster[0]}
  [649] = {fatherId=frmaster[0]}
  [650] = {fatherId=frmaster[0]}
  [651] = {fatherId=frmaster[0]}
  [652] = {fatherId=frmaster[0]}
  [653] = {fatherId=frmaster[0]}
  [654] = {fatherId=frmaster[0]}
  [655] = {fatherId=frmaster[0]}
  [656] = {fatherId=frmaster[0]}
  [657] = {fatherId=frmaster[0]}
  [658] = {fatherId=frmaster[0]}
  [659] = {fatherId=frmaster[0]}
  [660] = {fatherId=frmaster[0]}
  [661] = {fatherId=frmaster[0]}
  [662] = {fatherId=frmaster[0]}
  [663] = {fatherId=frmaster[0]}
  [664] = {fatherId=frmaster[0]}
  [665] = {fatherId=frmaster[0]}
  [666] = {fatherId=frmaster[0]}
  [667] = {fatherId=frmaster[0]}
  [668] = {fatherId=frmaster[0]}
  [669] = {fatherId=frmaster[0]}
  [670] = {fatherId=frmaster[0]}
  [671] = {fatherId=frmaster[0]}
  [672] = {fatherId=frmaster[0]}
  [673] = {fatherId=frmaster[0]}
  [674] = {fatherId=frmaster[0]}
  [675] = {fatherId=frmaster[0]}
  [676] = {fatherId=frmaster[0]}
  [677] = {fatherId=frmaster[0]}
  [678] = {fatherId=frmaster[0]}
  [679] = {fatherId=frmaster[0]}
  [680] = {fatherId=frmaster[0]}
  [681] = {fatherId=frmaster[0]}
  [682] = {fatherId=frmaster[0]}
  [683] = {fatherId=frmaster[0]}
  [684] = {fatherId=frmaster[0]}
  [685] = {fatherId=frmaster[0]}
  [686] = {fatherId=frmaster[0]}
  [687] = {fatherId=frmaster[0]}
  [688] = {fatherId=frmaster[0]}
  [689] = {fatherId=frmaster[0]}
  [690] = {fatherId=frmaster[0]}
  [691] = {fatherId=frmaster[0]}
  [692] = {fatherId=frmaster[0]}
  [693] = {fatherId=frmaster[0]}
  [694] = {fatherId=frmaster[0]}
  [695] = {fatherId=frmaster[0]}
  [696] = {fatherId=frmaster[0]}
  [697] = {fatherId=frmaster[0]}
  [698] = {fatherId=frmaster[0]}
  [699] = {fatherId=frmaster[0]}
  [700] = {fatherId=frmaster[0]}
  [701] = {fatherId=frmaster[0]}
  [702] = {fatherId=frmaster[0]}
  [703] = {fatherId=frmaster[0]}
  [704] = {fatherId=frmaster[0]}
  [705] = {fatherId=frmaster[0]}
  [706] = {fatherId=frmaster[0]}
  [707] = {fatherId=frmaster[0]}
  [708] = {fatherId=frmaster[0]}
  [709] = {fatherId=frmaster[0]}
  [710] = {fatherId=frmaster[0]}
  [711] = {fatherId=frmaster[0]}
  [712] = {fatherId=frmaster[0]}
  [713] = {fatherId=frmaster[0]}
  [714] = {fatherId=frmaster[0]}
  [715] = {fatherId=frmaster[0]}
  [716] = {fatherId=frmaster[0]}
  [717] = {fatherId=frmaster[0]}
  [718] = {fatherId=frmaster[0]}
  [719] = {fatherId=frmaster[0]}
  [720] = {fatherId=frmaster[0]}
  [721] = {fatherId=frmaster[0]}
  [722] = {fatherId=frmaster[0]}
  [723] = {fatherId=frmaster[0]}
  [724] = {fatherId=frmaster[0]}
  [725] = {fatherId=frmaster[0]}
  [726] = {fatherId=frmaster[0]}
  [727] = {fatherId=frmaster[0]}
  [728] = {fatherId=frmaster[0]}
  [729] = {fatherId=frmaster[0]}
  [730] = {fatherId=frmaster[0]}
  [731] = {fatherId=frmaster[0]}
  [732] = {fatherId=frmaster[0]}
  [733] = {fatherId=frmaster[0]}
  [734] = {fatherId=frmaster[0]}
  [735] = {fatherId=frmaster[0]}
  [736] = {fatherId=frmaster[0]}
  [737] = {fatherId=frmaster[0]}
  [738] = {fatherId=frmaster[0]}
  [739] = {fatherId=frmaster[0]}
  [740] = {fatherId=frmaster[0]}
  [741] = {fatherId=frmaster[0]}
  [742] = {fatherId=frmaster[0]}
  [743] = {fatherId=frmaster[0]}
  [744] = {fatherId=frmaster[0]}
  [745] = {fatherId=frmaster[0]}
  [746] = {fatherId=frmaster[0]}
  [747] = {fatherId=frmaster[0]}
  [748] = {fatherId=frmaster[0]}
  [749] = {fatherId=frmaster[0]}
  [750] = {fatherId=frmaster[0]}
  [751] = {fatherId=frmaster[0]}
  [752] = {fatherId=frmaster[0]}
  [753] = {fatherId=frmaster[0]}
  [754] = {fatherId=frmaster[0]}
  [755] = {fatherId=frmaster[0]}
  [756] = {fatherId=frmaster[0]}
  [757] = {fatherId=frmaster[0]}
  [758] = {fatherId=frmaster[0]}
  [759] = {fatherId=frmaster[0]}
  [760] = {fatherId=frmaster[0]}
  [761] = {fatherId=frmaster[0]}
  [762] = {fatherId=frmaster[0]}
  [763] = {fatherId=frmaster[0]}
  [764] = {fatherId=frmaster[0]}
  [765] = {fatherId=frmaster[0]}
  [766] = {fatherId=frmaster[0]}
  [767] = {fatherId=frmaster[0]}
  [768] = {fatherId=frmaster[0]}
  [769] = {fatherId=frmaster[0]}
  [770] = {fatherId=frmaster[0]}
  [771] = {fatherId=frmaster[0]}
  [772] = {fatherId=frmaster[0]}
  [773] = {fatherId=frmaster[0]}
  [774] = {fatherId=frmaster[0]}
  [775] = {fatherId=frmaster[0]}
  [776] = {fatherId=frmaster[0]}
  [777] = {fatherId=frmaster[0]}
  [778] = {fatherId=frmaster[0]}
  [779] = {fatherId=frmaster[0]}
  [780] = {fatherId=frmaster[0]}
  [781] = {fatherId=frmaster[0]}
  [782] = {fatherId=frmaster[0]}
  [783] = {fatherId=frmaster[0]}
  [784] = {fatherId=frmaster[0]}
  [785] = {fatherId=frmaster[0]}
  [786] = {fatherId=frmaster[0]}
  [787] = {fatherId=frmaster[0]}
  [788] = {fatherId=frmaster[0]}
  [789] = {fatherId=frmaster[0]}
  [790] = {fatherId=frmaster[0]}
  [791] = {fatherId=frmaster[0]}
  [792] = {fatherId=frmaster[0]}
  [793] = {fatherId=frmaster[0]}
  [794] = {fatherId=frmaster[0]}
  [795] = {fatherId=frmaster[0]}
  [796] = {fatherId=frmaster[0]}
  [797] = {fatherId=frmaster[0]}
  [798] = {fatherId=frmaster[0]}
  [799] = {fatherId=frmaster[0]}
  [800] = {fatherId=frmaster[0]}
  [801] = {fatherId=frmaster[0]}
  [802] = {fatherId=frmaster[0]}
  [803] = {fatherId=frmaster[0]}
  [804] = {fatherId=frmaster[0]}
  [805] = {fatherId=frmaster[0]}
  [806] = {fatherId=frmaster[0]}
  [807] = {fatherId=frmaster[0]}
  [808] = {fatherId=frmaster[0]}
  [809] = {fatherId=frmaster[0]}
  [810] = {fatherId=frmaster[0]}
  [811] = {fatherId=frmaster[0]}
  [812] = {fatherId=frmaster[0]}
  [813] = {fatherId=frmaster[0]}
  [814] = {fatherId=frmaster[0]}
  [815] = {fatherId=frmaster[0]}
  [816] = {fatherId=frmaster[0]}
  [817] = {fatherId=frmaster[0]}
  [818] = {fatherId=frmaster[0]}
  [819] = {fatherId=frmaster[0]}
  [820] = {fatherId=frmaster[0]}
  [821] = {fatherId=frmaster[0]}
  [822] = {fatherId=frmaster[0]}
  [823] = {fatherId=frmaster[0]}
  [824] = {fatherId=frmaster[0]}
  [825] = {fatherId=frmaster[0]}
  [826] = {fatherId=frmaster[0]}
  [827] = {fatherId=frmaster[0]}
  [828] = {fatherId=frmaster[0]}
  [829] = {fatherId=frmaster[0]}
  [830] = {fatherId=frmaster[0]}
  [831] = {fatherId=frmaster[0]}
  [832] = {fatherId=frmaster[0]}
  [833] = {fatherId=frmaster[0]}
  [834] = {fatherId=frmaster[0]}
  [835] = {fatherId=frmaster[0]}
  [836] = {fatherId=frmaster[0]}
  [837] = {fatherId=frmaster[0]}
  [838] = {fatherId=frmaster[0]}
  [839] = {fatherId=frmaster[0]}
  [840] = {fatherId=frmaster[0]}
  [841] = {fatherId=frmaster[0]}
  [842] = {fatherId=frmaster[0]}
  [843] = {fatherId=frmaster[0]}
  [844] = {fatherId=frmaster[0]}
  [845] = {fatherId=frmaster[0]}
  [846] = {fatherId=frmaster[0]}
  [847] = {fatherId=frmaster[0]}
  [848] = {fatherId=frmaster[0]}
  [849] = {fatherId=frmaster[0]}
  [850] = {fatherId=frmaster[0]}
  [851] = {fatherId=frmaster[0]}
  [852] = {fatherId=frmaster[0]}
  [853] = {fatherId=frmaster[0]}
  [854] = {fatherId=frmaster[0]}
  [855] = {fatherId=frmaster[0]}
  [856] = {fatherId=frmaster[0]}
  [857] = {fatherId=frmaster[0]}
  [858] = {fatherId=frmaster[0]}
  [859] = {fatherId=frmaster[0]}
  [860] = {fatherId=frmaster[0]}
  [861] = {fatherId=frmaster[0]}
  [862] = {fatherId=frmaster[0]}
  [863] = {fatherId=frmaster[0]}
  [864] = {fatherId=frmaster[0]}
  [865] = {fatherId=frmaster[0]}
  [866] = {fatherId=frmaster[0]}
  [867] = {fatherId=frmaster[0]}
  [868] = {fatherId=frmaster[0]}
  [869] = {fatherId=frmaster[0]}
  [870] = {fatherId=frmaster[0]}
  [871] = {fatherId=frmaster[0]}
  [872] = {fatherId=frmaster[0]}
  [873] = {fatherId=frmaster[0]}
  [874] = {fatherId=frmaster[0]}
  [875] = {fatherId=frmaster[0]}
  [876] = {fatherId=frmaster[0]}
  [877] = {fatherId=frmaster[0]}
  [878] = {fatherId=frmaster[0]}
  [879] = {fatherId=frmaster[0]}
  [880] = {fatherId=frmaster[0]}
  [881] = {fatherId=frmaster[0]}
  [882] = {fatherId=frmaster[0]}
  [883] = {fatherId=frmaster[0]}
  [884] = {fatherId=frmaster[0]}
  [885] = {fatherId=frmaster[0]}
  [886] = {fatherId=frmaster[0]}
  [887] = {fatherId=frmaster[0]}
  [888] = {fatherId=frmaster[0]}
  [889] = {fatherId=frmaster[0]}
  [890] = {fatherId=frmaster[0]}
  [891] = {fatherId=frmaster[0]}
  [892] = {fatherId=frmaster[0]}
  [893] = {fatherId=frmaster[0]}
  [894] = {fatherId=frmaster[0]}
  [895] = {fatherId=frmaster[0]}
  [896] = {fatherId=frmaster[0]}
  [897] = {fatherId=frmaster[0]}
  [898] = {fatherId=frmaster[0]}
  [899] = {fatherId=frmaster[0]}
pointRx pt1 = {fatherId=world[0]}
pointRx pt2 = {fatherId=world[0]}
pointRx pt3 = {fatherId=world[0]}
string sItem = "1点"
string sList[314]
  [0] = "1点"
  [1] = "2点"
  [2] = "3点"
  [3] = "4点"
  [4] = "5点"
  [5] = "6点"
  [6] = "7点"
  [7] = "8点"
  [8] = "9点"
  [9] = "10点"
  [10] = "11点"
  [11] = "12点"
  [12] = "13点"
  [13] = "14点"
  [14] = "15点"
  [15] = "16点"
  [16] = "17点"
  [17] = "18点"
  [18] = "19点"
  [19] = "20点"
  [20] = "21点"
  [21] = "22点"
  [22] = "23点"
  [23] = "24点"
  [24] = "25点"
  [25] = "26点"
  [26] = "27点"
  [27] = "28点"
  [28] = "29点"
  [29] = "30点"
  [30] = "31点"
  [31] = "32点"
  [32] = "33点"
  [33] = "34点"
  [34] = "35点"
  [35] = "36点"
  [36] = "37点"
  [37] = "38点"
  [38] = "39点"
  [39] = "40点"
  [40] = "41点"
  [41] = "42点"
  [42] = "43点"
  [43] = "44点"
  [44] = "45点"
  [45] = "46点"
  [46] = "47点"
  [47] = "48点"
  [48] = "49点"
  [49] = "50点"
  [50] = "51点"
  [51] = "52点"
  [52] = "53点"
  [53] = "54点"
  [54] = "55点"
  [55] = "56点"
  [56] = "57点"
  [57] = "58点"
  [58] = "59点"
  [59] = "60点"
  [60] = "61点"
  [61] = "62点"
  [62] = "63点"
  [63] = "64点"
  [64] = "65点"
  [65] = "66点"
  [66] = "67点"
  [67] = "68点"
  [68] = "69点"
  [69] = "70点"
  [70] = "71点"
  [71] = "72点"
  [72] = "73点"
  [73] = "74点"
  [74] = "75点"
  [75] = "76点"
  [76] = "77点"
  [77] = "78点"
  [78] = "79点"
  [79] = "80点"
  [80] = "81点"
  [81] = "82点"
  [82] = "83点"
  [83] = "84点"
  [84] = "85点"
  [85] = "86点"
  [86] = "87点"
  [87] = "88点"
  [88] = "89点"
  [89] = "90点"
  [90] = "91点"
  [91] = "92点"
  [92] = "93点"
  [93] = "94点"
  [94] = "95点"
  [95] = "96点"
  [96] = "97点"
  [97] = "98点"
  [98] = "99点"
  [99] = "100点"
  [100] = "101点"
  [101] = "102点"
  [102] = "103点"
  [103] = "104点"
  [104] = "105点"
  [105] = "106点"
  [106] = "107点"
  [107] = "108点"
  [108] = "109点"
  [109] = "110点"
  [110] = "111点"
  [111] = "112点"
  [112] = "113点"
  [113] = "114点"
  [114] = "115点"
  [115] = "116点"
  [116] = "117点"
  [117] = "118点"
  [118] = "119点"
  [119] = "120点"
  [120] = "121点"
  [121] = "122点"
  [122] = "123点"
  [123] = "124点"
  [124] = "125点"
  [125] = "126点"
  [126] = "127点"
  [127] = "128点"
  [128] = "129点"
  [129] = "130点"
  [130] = "131点"
  [131] = "132点"
  [132] = "133点"
  [133] = "134点"
  [134] = "135点"
  [135] = "136点"
  [136] = "137点"
  [137] = "138点"
  [138] = "139点"
  [139] = "140点"
  [140] = "141点"
  [141] = "142点"
  [142] = "143点"
  [143] = "144点"
  [144] = "145点"
  [145] = "146点"
  [146] = "147点"
  [147] = "148点"
  [148] = "149点"
  [149] = "150点"
  [150] = "151点"
  [151] = "152点"
  [152] = "153点"
  [153] = "154点"
  [154] = "155点"
  [155] = "156点"
  [156] = "157点"
  [157] = "158点"
  [158] = "159点"
  [159] = "160点"
  [160] = "161点"
  [161] = "162点"
  [162] = "163点"
  [163] = "164点"
  [164] = "165点"
  [165] = "166点"
  [166] = "167点"
  [167] = "168点"
  [168] = "169点"
  [169] = "170点"
  [170] = "171点"
  [171] = "172点"
  [172] = "173点"
  [173] = "174点"
  [174] = "175点"
  [175] = "176点"
  [176] = "177点"
  [177] = "178点"
  [178] = "179点"
  [179] = "180点"
  [180] = "181点"
  [181] = "182点"
  [182] = "183点"
  [183] = "184点"
  [184] = "185点"
  [185] = "186点"
  [186] = "187点"
  [187] = "188点"
  [188] = "189点"
  [189] = "190点"
  [190] = "191点"
  [191] = "192点"
  [192] = "193点"
  [193] = "194点"
  [194] = "195点"
  [195] = "196点"
  [196] = "197点"
  [197] = "198点"
  [198] = "199点"
  [199] = "200点"
  [200] = "201点"
  [201] = "202点"
  [202] = "203点"
  [203] = "204点"
  [204] = "205点"
  [205] = "206点"
  [206] = "207点"
  [207] = "208点"
  [208] = "209点"
  [209] = "210点"
  [210] = "211点"
  [211] = "212点"
  [212] = "213点"
  [213] = "214点"
  [214] = "215点"
  [215] = "216点"
  [216] = "217点"
  [217] = "218点"
  [218] = "219点"
  [219] = "220点"
  [220] = "221点"
  [221] = "222点"
  [222] = "223点"
  [223] = "224点"
  [224] = "225点"
  [225] = "226点"
  [226] = "227点"
  [227] = "228点"
  [228] = "229点"
  [229] = "230点"
  [230] = "231点"
  [231] = "232点"
  [232] = "233点"
  [233] = "234点"
  [234] = "235点"
  [235] = "236点"
  [236] = "237点"
  [237] = "238点"
  [238] = "239点"
  [239] = "240点"
  [240] = "241点"
  [241] = "242点"
  [242] = "243点"
  [243] = "244点"
  [244] = "245点"
  [245] = "246点"
  [246] = "247点"
  [247] = "248点"
  [248] = "249点"
  [249] = "250点"
  [250] = "251点"
  [251] = "252点"
  [252] = "253点"
  [253] = "254点"
  [254] = "255点"
  [255] = "256点"
  [256] = "257点"
  [257] = "258点"
  [258] = "259点"
  [259] = "260点"
  [260] = "261点"
  [261] = "262点"
  [262] = "263点"
  [263] = "264点"
  [264] = "265点"
  [265] = "266点"
  [266] = "267点"
  [267] = "268点"
  [268] = "269点"
  [269] = "270点"
  [270] = "271点"
  [271] = "272点"
  [272] = "273点"
  [273] = "274点"
  [274] = "275点"
  [275] = "276点"
  [276] = "277点"
  [277] = "278点"
  [278] = "279点"
  [279] = "280点"
  [280] = "281点"
  [281] = "282点"
  [282] = "283点"
  [283] = "284点"
  [284] = "285点"
  [285] = "286点"
  [286] = "287点"
  [287] = "288点"
  [288] = "289点"
  [289] = "290点"
  [290] = "291点"
  [291] = "292点"
  [292] = "293点"
  [293] = "294点"
  [294] = "295点"
  [295] = "296点"
  [296] = "297点"
  [297] = "298点"
  [298] = "299点"
  [299] = "300点"
  [300] = "301点"
  [301] = "302点"
  [302] = "303点"
  [303] = "304点"
  [304] = "305点"
  [305] = "306点"
  [306] = "307点"
  [307] = "308点"
  [308] = "309点"
  [309] = "310点"
  [310] = "311点"
  [311] = "312点"
  [312] = "313点"
  [313] = "314点"
string sListItemValue[3]
  [0] = "0   "
  [1] = "0   "
  [2] = "0   "
string sMsg[8]
string sParameter[3]
  [0] = "X        :0         "
  [1] = "Y        :0         "
  [2] = "Z        :0         "
tool t1 = {fatherId=flange[0], ioLink=valve1}
tool t2 = {x=0.1, fatherId=flange[0], ioLink=valve1}
trsf trOffset
